(* Logix 5000 project; controller PBS_Perfusion vendor 1 type 14 code 217 rev 32.14; software revision 32.03; part 22 of 27 *)
(* tags used below, declared in another part *)
   Inp_SpeedFdbk : REAL;   // Speed Feedbak in Drive Units (typ. 0-32767 = 0 to max freq.)
   Inp_Datalink : REAL;   // Auxiliary Signal (datalink) Input in Drive (raw) Units
   Inp_Ready : BOOL;   // 1=Drive is ready to run
   Inp_Running : BOOL;   // 1=Drive is Running (active)
   Inp_CommandDir : BOOL;   // 1=Drive is commanded Forward, 0=Drive is commanded Reverse
   Inp_ActualDir : BOOL;   // 1=Drive is running Forward, 0=Drive is running Reverse
   Inp_Accelerating : BOOL;   // 1=Drive is accelerating
   Inp_Decelerating : BOOL;   // 1=Drive is decelerating
   Inp_Alarm : BOOL;   // 1=Drive has an Alarm Condition (see drive display or manual)
   Inp_Faulted : BOOL;   // 1=Drive has Faulted (see drive display or manual)
   Inp_AtSpeed : BOOL;   // 1=Drive is at commanded speed
   Inp_FwdPermOK : BOOL;   // 1=Permissives OK, drive can start Forward
   Inp_FwdNBPermOK : BOOL;   // 1=Non-Bypassable Permissives OK, drive can start Forward
   Inp_RevPermOK : BOOL;   // 1=Permissives OK, drive can start Reverse
   Inp_RevNBPermOK : BOOL;   // 1=Non-Bypassable Permissives OK, motor can start Reverse
   Inp_IntlkOK : BOOL;   // 1=Interlocks OK, drive can start/run
   Inp_NBIntlkOK : BOOL;   // 1=Non-Bypassable Interlocks OK, drive can start/run
   Inp_IntlkAvail : BOOL;   // 1 = Interlock Availibility OK
   Inp_IOFault : BOOL;   // Input Communication Status 0=OK, 1=fail
   Inp_Sim : BOOL;   // 1=Simulate working drive; 0=Start/Stop/ Monitor actual drive
   Inp_OvrdCmd : DINT;   // Override Command: 0=None, 1=Stop, 2=Start Fwd 3=Start Rev
   Inp_OvrdSpeed : REAL;   // Value to set Speed Reference in Override Mode (SpeedRef EU)
   Inp_OvrdOutDatalink : REAL;   // Value to set Output Datalink in Override Mode (OutDatalink EU)
   Inp_Reset : BOOL;   // 1=Reset Shed Latches and Cleared Alarms
   Cfg_HasReverse : BOOL;   // 1=Drive can be run reverse, 0=Forward only
   Cfg_HasJog : BOOL;   // 1=Drive Jog Command enabled/visible, 0=Drive Jog Command not allowed
   Cfg_AllowLocal : BOOL;   // 1=Allow Local Start/Stop without alarm, 0=Start/Stop from HMI/prog only
   Cfg_HasRunFdbk : BOOL;   // 1=Drive provides feedback signal on Inp_Running when running
   Cfg_UseRunFdbk : BOOL;   // 1=Drive run feedback should be used for failure checking
   Cfg_HasSpeedFdbk : BOOL;   // 1=Drive provides speed feedback on Inp_SpeedFdbk
   Cfg_UseSpeedFdbk : BOOL;   // 1=Drive speed determines running state, 0=state determined by drive Active input bit
   Cfg_HasInpDatalink : BOOL;   // 1=A signal is connected to Inp_Datalink
   Cfg_SetTrack : BOOL;   // 1=Settings track for unselected sources, 0=no tracking
   Cfg_SetTrackOvrdHand : BOOL;   // 1=Prog/Oper/Ext Settings track Override/Hand
   Cfg_OperStopPrio : BOOL;   // 1=OCmd_Stop any time, 0=OCmd_Stop only when Oper selected
   Cfg_ExtStopPrio : BOOL;   // 1=XCmd_Stop any time, 0=XCmd_Stop only when Ext selected
   Cfg_OCmdResets : BOOL;   // 1=New drive OCmd resets shed latches and cleared alarms, 0=OCmdReset req'd.
   Cfg_XCmdResets : BOOL;   // 1=New drive XCmd resets shed latches and cleared alarms, 0=XCmdReset req'd.
   Cfg_OvrdPermIntlk : BOOL;   // 1=Override ignores Bypassable Perm/ Intlk; 0=always use Perm/Intlk
   Cfg_ShedOnIOFault : BOOL;   // 1=Stop Motor and Alarm on I/O Fault; 0=Alarm only on I/O Fault
   Cfg_SimScaleEU : BOOL;   // 1=In simulation, scale Speed Ref EU to Speed Fdbk EU
   Cfg_SimScaleRaw : BOOL;   // 1=In simulation, scale Speed Ref EU to raw, then raw to Speed Fdbk EU
   Cfg_MaxSpdRef : REAL;   // Maximum Speed Reference in EU (for limiting)
   Cfg_SpeedRefRawMin : REAL;   // Speed Reference Minimum in Drive (raw) Units (for scaling)
   Cfg_SpeedRefRawMax : REAL;   // Speed Reference Maximum in Drive (raw) Units (for scaling)
   Cfg_SpeedRefEUMin : REAL;   // Speed Reference Minimum in Engineering Units (for scaling)
   Cfg_SpeedRefEUMax : REAL;   // Speed Reference Maximum in Engineering Units (for scaling)
   Cfg_SpeedFdbkRawMin : REAL;   // Speed Feedback Minimum in Drive (raw) Units (for scaling)
   Cfg_SpeedFdbkRawMax : REAL;   // Speed Feedback Maximum in Drive (raw) Units (for scaling)
   Cfg_SpeedFdbkEUMin : REAL;   // Speed Feedback Minimum in Engineering Units (for scaling)
   Cfg_SpeedFdbkEUMax : REAL;   // Speed Feedback Maximum in Engineering Units (for scaling)
   Cfg_InpDatalinkRawMin : REAL;   // Input Datalink Minimum in Drive (raw) Units (for scaling)
   Cfg_InpDatalinkRawMax : REAL;   // Input Datalink Maximum in Drive (raw) Units (for scaling)
   Cfg_InpDatalinkEUMin : REAL;   // Input Datalink Minimum in Engineering Units (for scaling)
   Cfg_InpDatalinkEUMax : REAL;   // Input Datalink Maximum in Engineering Units (for scaling)
   Cfg_OutDatalinkMin : REAL;   // Minimum Output Datalink in EU (for limiting)
   Cfg_OutDatalinkMax : REAL;   // Maximum Output Datalink in EU (for limiting)
   Cfg_SimRampT : REAL;   // Time to ramp speed fdbk when in Simulation (sec)
   PSet_SpeedRef : REAL;   // Program Setting of Speed Reference (EU)
   PSet_OutDatalink : REAL;   // Program Setting of Output Datalink (EU)
   XSet_SpeedRef : REAL;   // External Setting of Speed Reference (EU)
   XSet_OutDatalink : REAL;   // External Setting of Output Datalink (EU)
   PCmd_StartFwd : BOOL;   // Program Command to Start Drive Forward
   PCmd_StartRev : BOOL;   // Program Command to Start Drive Reverse
   PCmd_Stop : BOOL;   // Program Command to Stop Drive
   PCmd_Reset : BOOL;   // Program Command to Reset drive fault and all Alarms requiring Reset
   PCmd_FailToStartAck : ALIAS FOR FailToStart.PCmd_Ack;   // Program Command to Acknowledge Fail to Start Alarm
   PCmd_FailToStopAck : ALIAS FOR FailToStop.PCmd_Ack;   // Program Command to Acknowledge Fail to Stop Alarm
   PCmd_IntlkTripAck : ALIAS FOR IntlkTrip.PCmd_Ack;   // Program Command to Acknowledge Interlock Trip Alarm
   PCmd_DriveFaultAck : ALIAS FOR DriveFault.PCmd_Ack;   // Program Command to Acknowledge Drive Fault Alarm
   PCmd_IOFaultAck : ALIAS FOR IOFault.PCmd_Ack;   // Program Command to Acknowledge I/O Fault Alarm
   XCmd_StartFwd : BOOL;   // External Command to Start Drive Forward
   XCmd_StartRev : BOOL;   // External Command to Start Drive Reverse
   XCmd_Stop : BOOL;   // External Command to Stop Drive
   XCmd_JogFwd : BOOL;   // External Command to Jog Drive Forward
   XCmd_JogRev : BOOL;   // External Command to Jog Drive Reverse
   XCmd_Reset : BOOL;   // Ext Cmd to clear shed latches and cleared alarms
   Out_ClearFault : BOOL;   // 1=Attempt to clear Drive Fault
   Val_SpeedFdbk : REAL;   // Speed Feedback (actual) from drive
   Val_InpDatalink : REAL;   // Input Datalink value from drive
   Val_SpeedFdbkEUMin : REAL;   // Minimum of Speed Feedback = MIN (Cfg_SpeedFdbkEUMin, Cfg_SpeedFdbkEUMax)
   Val_SpeedFdbkEUMax : REAL;   // Maximum of Speed Feedback = MAX (Cfg_SpeedFdbkEUMin, Cfg_SpeedFdbkEUMax)
   Val_Fdbk : DINT;   // Device Feedback 0=Stopped, 1=Running Fwd 2=Running Rev 3=Accelerating 4=Decelerating
   Sts_StartingFwd : BOOL;   // 1=Drive requested to run forward and awaiting run feedback
   Sts_StartingRev : BOOL;   // 1=Drive requested to run reverse and awaiting run feedback
   Sts_RunningFwd : BOOL;   // 1=Drive requested to run and is confirmed running forward
   Sts_RunningRev : BOOL;   // 1=Drive requested to run and is confirmed running reverse
   Sts_CommandDir : BOOL;   // 1=Drive commanded to Forward, 0=Reverse
   Sts_ActualDir : BOOL;   // 1=Drive Actual direction is Forward, 0=Reverse
   Sts_Accel : BOOL;   // 1=Drive is Accelerating
   Sts_Decel : BOOL;   // 1=Drive is Decelerating
   Sts_NotReady : BOOL;   // 1=Drive is Not Ready (cannot be started) Check alarms, stops, faults
   Sts_Alarm : BOOL;   // 1=Drive has an Alarm (see drive display or manual)
   Sts_AtSpeed : BOOL;   // 1=Drive is running at reference speed
   Sts_Available : BOOL;   // 1=Drive available for control by automation (Prog)
   Sts_Bypass : BOOL;   // 1=Bypassable Interlocks and Permissives are Bypassed
   Sts_BypActive : BOOL;   // 1=Bypassing Active (Bypassed or Maintenance)
   Sts_NotRdy : BOOL;   // 1=Device Not Ready, see detail bits for reason
   Nrdy_CfgErr : BOOL;   // 1=Device Not Ready: Configuration Error
   Nrdy_DriveNR : BOOL;   // 1=Device Note Ready: Drive Not Ready
   Nrdy_Fail : BOOL;   // 1=Device Not Ready: Device Failure (Shed Requires Reset)
   Nrdy_Intlk : BOOL;   // 1=Device Not Ready: Interlock Not OK
   Nrdy_IOFault : BOOL;   // 1=Device Not Ready: I/O Fault (Shed Requires Reset)
   Nrdy_OoS : BOOL;   // 1=Device Not Ready: Device is Out of Service
   Nrdy_Perm : BOOL;   // 1=Device Not Ready: Permissive Not OK
   Nrdy_PrioStop : BOOL;   // 1=Device Not Ready: Oper/Ext Priority Stop Requires Reset
   Nrdy_Trip : BOOL;   // 1=Device not Ready: Deivce Tripped (Drive Fault)
   Sts_MaintByp : BOOL;   // 1=A Maintenance Bypass is Active, display icon
   Err_FdbkRaw : BOOL;   // 1=Erron in Config: Speed Fdbk Raw Min = Max
   Err_FdbkEU : BOOL;   // 1=Error in Config: Speed Fdbk EU Min = Max
   Err_RefEU : BOOL;   // 1=Error in Config: Speed Ref EU Min = Max
   Err_InpDLEU : BOOL;   // 1=Error in Config: Input Datalink EU Min = Max
   Sts_Hand : ALIAS FOR CmdSrc.Sts_Hand;
   Sts_OoS : ALIAS FOR CmdSrc.Sts_OoS;
   Sts_Maint : ALIAS FOR CmdSrc.Sts_Maint;
   Sts_Ovrd : ALIAS FOR CmdSrc.Sts_Ovrd;
   Sts_Prog : ALIAS FOR CmdSrc.Sts_Prog;
   Sts_Oper : ALIAS FOR CmdSrc.Sts_Oper;
   Sts_FailToStart : ALIAS FOR FailToStart.Inp;   // 1=Drive Failed to Start (One-Shot)
   Sts_FailToStop : ALIAS FOR FailToStop.Inp;   // 1=Drive Failed to Stop
   Sts_IntlkTrip : ALIAS FOR IntlkTrip.Inp;   // 1=Drive was stopped by an Interlock NOT OK (One-Shot)
   Sts_DriveFault : ALIAS FOR DriveFault.Inp;   // 1=Drive Fault (see drive display or manual)
   Sts_IOFault : ALIAS FOR IOFault.Inp;   // I/O Comm Fault Status (0=OK, 1=Bad)
   P_VSD : BOOL;   // Unique Parameter Name for auto - discovery
   CmdSrc : P_CmdSrc;   // Drive Mode Selection
   IOFault : P_Alarm;   // I/O Fault Alarm
   IntlkTrip : P_Alarm;   // Interlock Trip Alarm
   FailToStop : P_Alarm;   // Drive Failed to Stop Alarm
   FailToStart : P_Alarm;   // Drive Failed to Start Alarm
   Wrk_Run : BOOL;   // 1=Drive should be "running", 0=should be "stopped"
   Wrk_StartRetrigT : TIMER;   // Time to pulse start output on start command retrigger (Maint)
   Wrk_StopRetrigT : TIMER;   // Time to pulse stop output on stop command retrigger (Maint)
   Wrk_RunFdbk : BOOL;   // Run Feedback based on mode, simulation, etc. 1=running
   Wrk_Bypass : BOOL;   // Internal Bypassable Permissives and Interlocks are Bypassed flag
   DriveFault : P_Alarm;   // Drive Faulted Alarm
   Wrk_SpeedRef : REAL;   // Working copy of Speed Reference (for limiting)
   Wrk_Rev : BOOL;   // Working (internal) Direction 1=Reverse 0=Forward (default)
   Wrk_Jog : BOOL;   // 1=Jog Drive, 0=Drive not jogging
   Wrk_ResetT : TIMER;   // Reset Output Pulse Timer
   Wrk_ResetONS : BOOL;   // One-Shot to fire Reset Timer to ensure min. output ON time.
   Wrk_OutDatalink : REAL;   // Selected Output Datalink setting
   Wrk_StopT : TIMER;   // Stop Check Timer (for Fail to Stop)
   Wrk_StartT : TIMER;   // Start Check Timer (for Fail to Start)
   Wrk_Retrigger : BOOL;   // Maint Start issued while running or Stop while stopped
   Wrk_Step : REAL;   // Amount to change simulated Speed Fdbk this scan (ramp)
   Wrk_ScanTime : REAL;   // Seconds since previous scan
   Wrk_ScanT : TIMER;   // Scan Timer (milliseconds, always runs)
   Wrk_SimFdbkTgt : REAL;   // Speed Ref converted to Speed Fdbk units for simulation: target speed fdbk
   Wrk_JogT : TIMER;   // Jog Timer
   Wrk_SimScaleEUONS : BOOL;   // Cfg_SimScaleEU became true this scan
   Wrk_SimScaleRawONS : BOOL;   // Cfg_SimScaleRaw became true this scan
   Wrk_NotRdyONS : BOOL;   // Assert Stop on One-Shot of Sts_NotRdy
   Wrk_NotRdy : BOOL;   // Device Not Ready conditions excluding shed latches
   Wrk_StartInhT : TIMER;   // Local Start Inhibit Timer
   Wrk_StopInhT : TIMER;   // Local Stop Inhibit Timer
   Wrk_NoLongerSim : BOOL;   // Switched from Simulated to Real Drive this scan
   Wrk_Hand : BOOL;   // Perform Hand Mode alignment with actual device state
   Wrk_StartHornT : TIMER;   // Timer for audible alert or start
   Wrk_StartHorn : BOOL;   // 1=Sound audible prior to commanded motor start
   Wrk_RevPermOK : BOOL;   // Reverse Permissives and NB Permissive OK
   Wrk_FwdPermOK : BOOL;   // Forward Permissives and NB Permissive OK
   OCmd_ResetAckAll : BOOL;   // Oper Cmd to reset shed latches and cleared alarms, plus Acknowledge alarms
   OCmd_Reset : BOOL;   // Oper Cmd to clear shed latches and cleared alarms
   OCmd_JogRev : BOOL;   // Operator Command to Jog Drive Reverse (not cleared by instruction!)
   OCmd_JogFwd : BOOL;   // Operator Command to Jog Drive Forward (not cleared by instruction!)
   OCmd_Stop : BOOL;   // Operator Command to Stop Drive
   OCmd_StartRev : BOOL;   // Operator Command to Start Drive Reverse
   OCmd_StartFwd : BOOL;   // Operator Command to Start Drive Forward
   MCmd_Check : BOOL;   // Maintenance Command to Check (not bypass) all Interlocks and Permissives
   MCmd_Bypass : BOOL;   // Maintenance Command to Bypass all Bypassable Interlocks and Permissives
   OSet_OutDatalink : REAL;   // Operator Setting of Output Datalink (EU)
   OSet_SpeedRef : REAL;   // Operator Setting of Speed Reference (EU)
   ORdy_OSet : BOOL;   // 1=Ready for OSets (other than Speed Ref) (enables data entry fields)
   ORdy_SpeedRef : BOOL;   // 1=Ready for OSet_SpeedRef (enables data entry field)
   MRdy_Check : BOOL;   // 1=Ready for MCmd_Check (enables HMI button)
   MRdy_Bypass : BOOL;   // 1=Ready for MCmd_Bypass (enables HMI button)
   Wrk_ExtHas3 : BOOL;   // External has Output Datalink
   Wrk_ExtHas1 : BOOL;   // External has Commands
   Wrk_ExtHas0 : BOOL;   // External has Speed Reference
   Wrk_ProgHas3 : BOOL;   // Program has Output Datalink
   Wrk_ProgHas1 : BOOL;   // Program has Commands
   Wrk_ProgHas0 : BOOL;   // Program has Speed Reference
   Wrk_OperHas3 : BOOL;   // Operator has Output Datalink
   Wrk_OperHas1 : BOOL;   // Operator has Commands
   Wrk_OperHas0 : BOOL;   // Operator has Speed Reference
   ONS : DINT[3];
   REAL : DINT;
(* P_VSD, continued *)

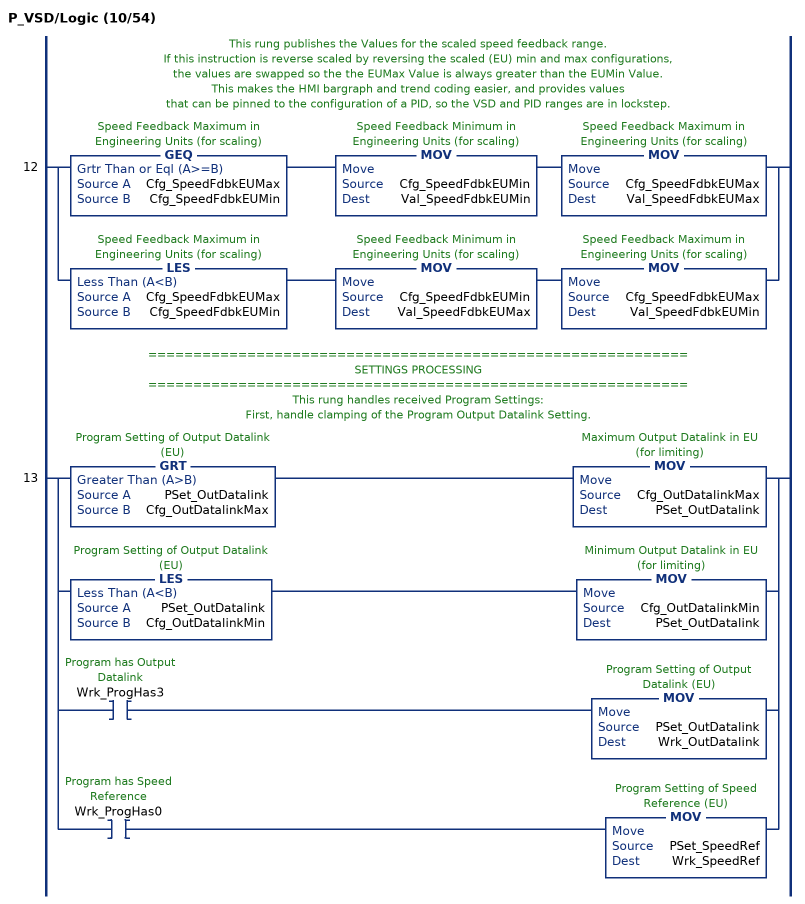
   [picture p487: P_VSD/Logic rungs 12-13]
   // This rung publishes the Values for the scaled speed feedback range.
   // If this instruction is reverse scaled by reversing the scaled (EU) min and max configurations,
   // the values are swapped so the the EUMax Value is always greater than the EUMin Value.
   // This makes the HMI bargraph and trend coding easier, and provides values
   // that can be pinned to the configuration of a PID, so the VSD and PID ranges are in lockstep.
   12: [GEQ(Cfg_SpeedFdbkEUMax,Cfg_SpeedFdbkEUMin) MOV(Cfg_SpeedFdbkEUMin,Val_SpeedFdbkEUMin) MOV(Cfg_SpeedFdbkEUMax,Val_SpeedFdbkEUMax) ,LES(Cfg_SpeedFdbkEUMax,Cfg_SpeedFdbkEUMin) MOV(Cfg_SpeedFdbkEUMin,Val_SpeedFdbkEUMax) MOV(Cfg_SpeedFdbkEUMax,Val_SpeedFdbkEUMin) ];
   // ============================================================
   // SETTINGS PROCESSING
   // ============================================================
   // This rung handles received Program Settings:
   // First, handle clamping of the Program Output Datalink Setting.
   13: [GRT(PSet_OutDatalink,Cfg_OutDatalinkMax) MOV(Cfg_OutDatalinkMax,PSet_OutDatalink) ,LES(PSet_OutDatalink,Cfg_OutDatalinkMin) MOV(Cfg_OutDatalinkMin,PSet_OutDatalink) ,XIC(Wrk_ProgHas3) MOV(PSet_OutDatalink,Wrk_OutDatalink) ,XIC(Wrk_ProgHas0) MOV(PSet_SpeedRef,Wrk_SpeedRef) ];
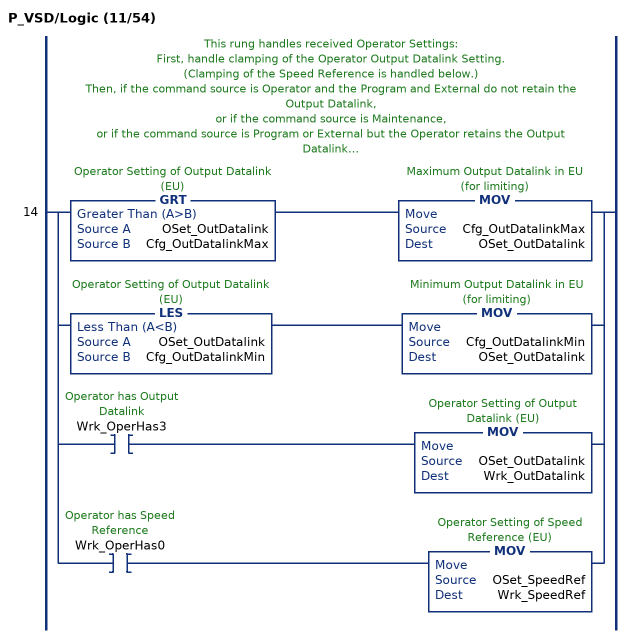
   // This rung handles received Operator Settings:
   // First, handle clamping of the Operator Output Datalink Setting.
   // (Clamping of the Speed Reference is handled below.)
   // Then, if the command source is Operator and the Program and External do not retain the Output Datalink,
   // or if the command source is Maintenance,
   // or if the command source is Program or External but the Operator retains the Output Datalink,
   // use the Operator Setting for the Output Datalink.
   // The Operator Setting for the Speed Reference is handled similarly.
   // #####  Changed P_Mode to P_CmdSrc. Added External Command Source and Commands.  #####
   14: [GRT(OSet_OutDatalink,Cfg_OutDatalinkMax) MOV(Cfg_OutDatalinkMax,OSet_OutDatalink) ,LES(OSet_OutDatalink,Cfg_OutDatalinkMin) MOV(Cfg_OutDatalinkMin,OSet_OutDatalink) ,XIC(Wrk_OperHas3) MOV(OSet_OutDatalink,Wrk_OutDatalink) ,XIC(Wrk_OperHas0) MOV(OSet_SpeedRef,Wrk_SpeedRef) ];
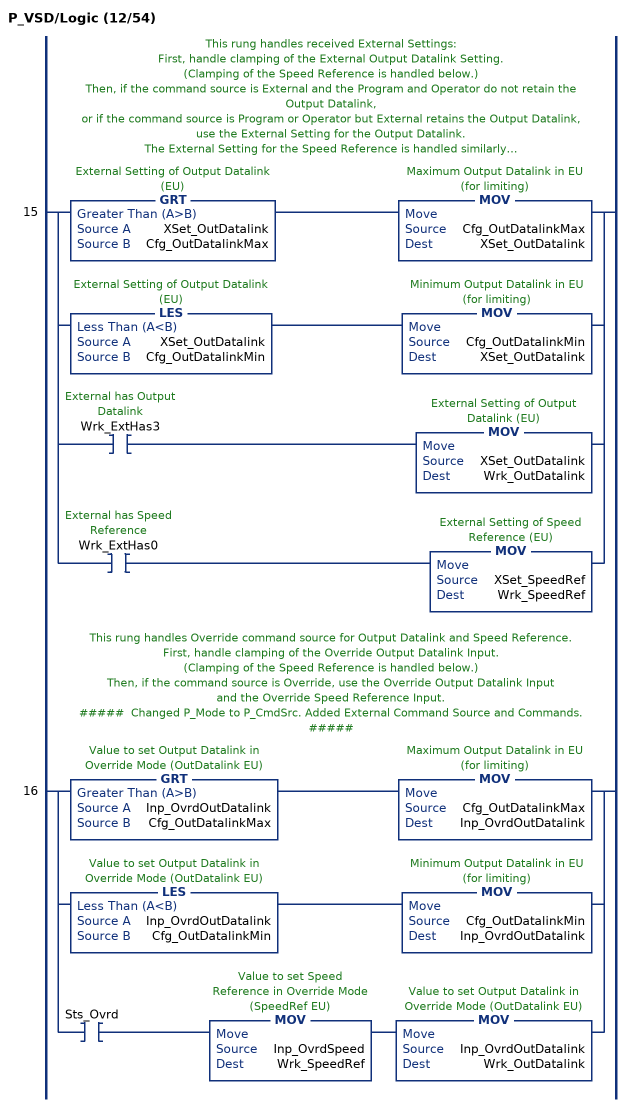
   // This rung handles received External Settings:
   // First, handle clamping of the External Output Datalink Setting.
   // (Clamping of the Speed Reference is handled below.)
   // Then, if the command source is External and the Program and Operator do not retain the Output Datalink,
   // or if the command source is Program or Operator but External retains the Output Datalink,
   // use the External Setting for the Output Datalink.
   // The External Setting for the Speed Reference is handled similarly.
   // #####  Changed P_Mode to P_CmdSrc. Added External Command Source and Commands.  #####
   15: [GRT(XSet_OutDatalink,Cfg_OutDatalinkMax) MOV(Cfg_OutDatalinkMax,XSet_OutDatalink) ,LES(XSet_OutDatalink,Cfg_OutDatalinkMin) MOV(Cfg_OutDatalinkMin,XSet_OutDatalink) ,XIC(Wrk_ExtHas3) MOV(XSet_OutDatalink,Wrk_OutDatalink) ,XIC(Wrk_ExtHas0) MOV(XSet_SpeedRef,Wrk_SpeedRef) ];
   // This rung handles Override command source for Output Datalink and Speed Reference.
   // First, handle clamping of the Override Output Datalink Input.
   // (Clamping of the Speed Reference is handled below.)
   // Then, if the command source is Override, use the Override Output Datalink Input
   // and the Override Speed Reference Input.
   // #####  Changed P_Mode to P_CmdSrc. Added External Command Source and Commands.  #####
   16: [GRT(Inp_OvrdOutDatalink,Cfg_OutDatalinkMax) MOV(Cfg_OutDatalinkMax,Inp_OvrdOutDatalink) ,LES(Inp_OvrdOutDatalink,Cfg_OutDatalinkMin) MOV(Cfg_OutDatalinkMin,Inp_OvrdOutDatalink) ,XIC(Sts_Ovrd) MOV(Inp_OvrdSpeed,Wrk_SpeedRef) MOV(Inp_OvrdOutDatalink,Wrk_OutDatalink) ];
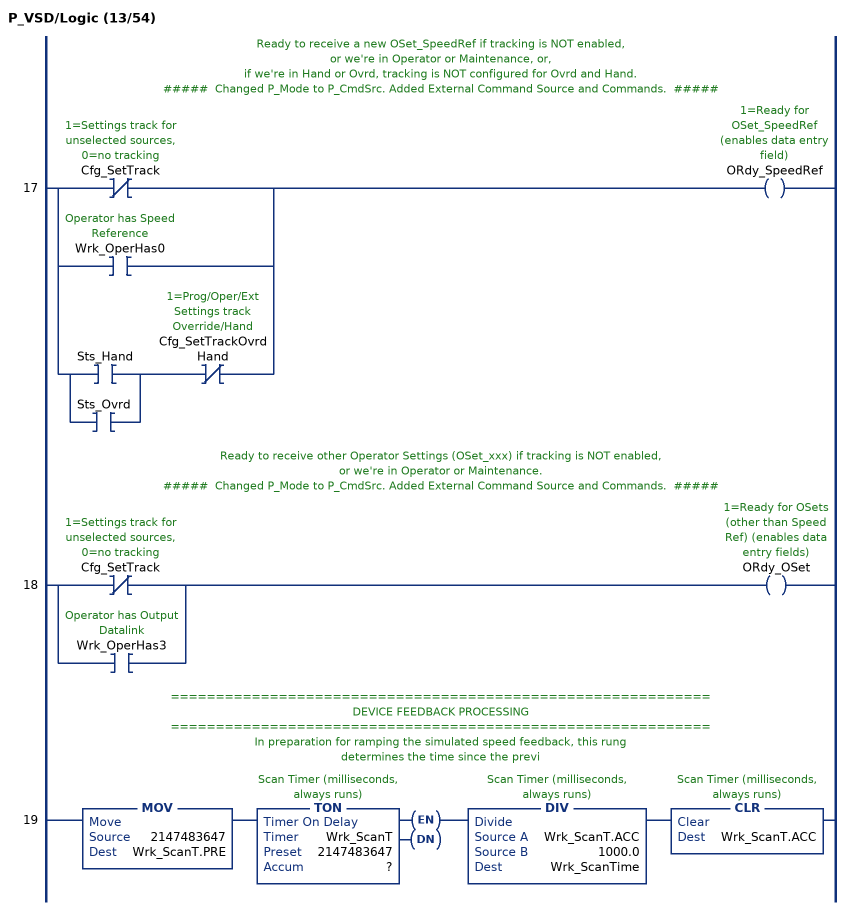
   // Ready to receive a new OSet_SpeedRef if tracking is NOT enabled,
   // or we're in Operator or Maintenance, or,
   // if we're in Hand or Ovrd, tracking is NOT configured for Ovrd and Hand.
   // #####  Changed P_Mode to P_CmdSrc. Added External Command Source and Commands.  #####
   17: [XIO(Cfg_SetTrack) ,XIC(Wrk_OperHas0) ,[XIC(Sts_Hand) ,XIC(Sts_Ovrd) ] XIO(Cfg_SetTrackOvrdHand) ]OTE(ORdy_SpeedRef);
   // Ready to receive other Operator Settings (OSet_xxx) if tracking is NOT enabled,
   // or we're in Operator or Maintenance.
   // #####  Changed P_Mode to P_CmdSrc. Added External Command Source and Commands.  #####
   18: [XIO(Cfg_SetTrack) ,XIC(Wrk_OperHas3) ]OTE(ORdy_OSet);
   // ============================================================
   // DEVICE FEEDBACK PROCESSING
   // ============================================================
   // In preparation for ramping the simulated speed feedback, this rung
   // determines the time since the previ
   19: MOV(2147483647,Wrk_ScanT.PRE)TON(Wrk_ScanT,?,?)DIV(Wrk_ScanT.ACC,1000.0,Wrk_ScanTime)CLR(Wrk_ScanT.ACC);
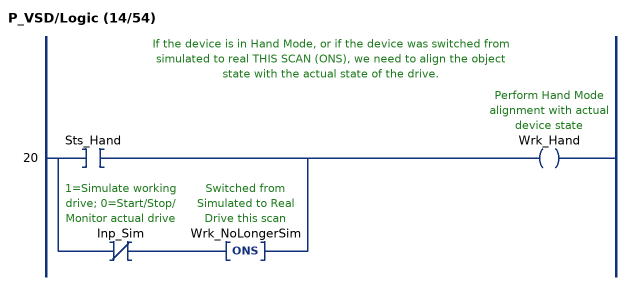
   // If the device is in Hand Mode, or if the device was switched from
   // simulated to real THIS SCAN (ONS), we need to align the object
   // state with the actual state of the drive.
   20: [XIC(Sts_Hand) ,XIO(Inp_Sim) ONS(Wrk_NoLongerSim) ]OTE(Wrk_Hand);
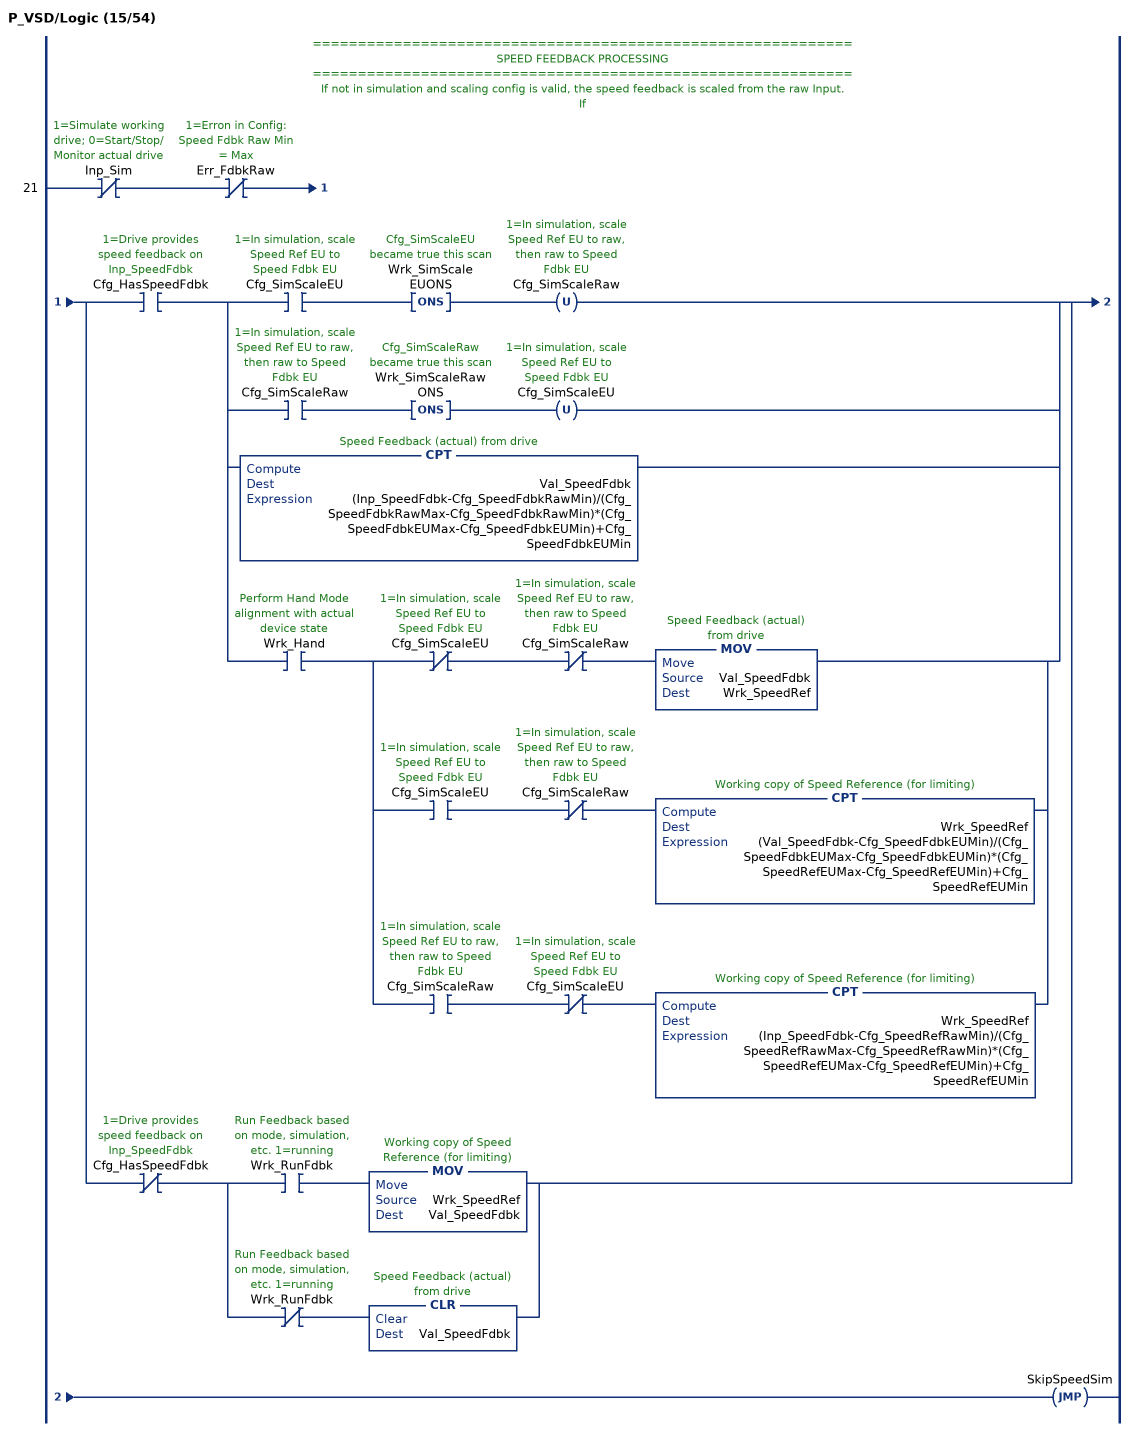
   // ============================================================
   // SPEED FEEDBACK PROCESSING
   // ============================================================
   // If not in simulation and scaling config is valid, the speed feedback is scaled from the raw Input.
   // If
   21: XIO(Inp_Sim)XIO(Err_FdbkRaw)[XIC(Cfg_HasSpeedFdbk) [XIC(Cfg_SimScaleEU) ONS(Wrk_SimScaleEUONS) OTU(Cfg_SimScaleRaw) ,XIC(Cfg_SimScaleRaw) ONS(Wrk_SimScaleRawONS) OTU(Cfg_SimScaleEU) ,CPT(Val_SpeedFdbk,(Inp_SpeedFdbk-Cfg_SpeedFdbkRawMin)/(Cfg_SpeedFdbkRawMax-Cfg_SpeedFdbkRawMin)*(Cfg_SpeedFdbkEUMax-Cfg_SpeedFdbkEUMin)+Cfg_SpeedFdbkEUMin) ,XIC(Wrk_Hand) [XIO(Cfg_SimScaleEU) XIO(Cfg_SimScaleRaw) MOV(Val_SpeedFdbk,Wrk_SpeedRef) ,XIC(Cfg_SimScaleEU) XIO(Cfg_SimScaleRaw) CPT(Wrk_SpeedRef,(Val_SpeedFdbk-Cfg_SpeedFdbkEUMin)/(Cfg_SpeedFdbkEUMax-Cfg_SpeedFdbkEUMin)*(Cfg_SpeedRefEUMax-Cfg_SpeedRefEUMin)+Cfg_SpeedRefEUMin) ,XIC(Cfg_SimScaleRaw) XIO(Cfg_SimScaleEU) CPT(Wrk_SpeedRef,(Inp_SpeedFdbk-Cfg_SpeedRefRawMin)/(Cfg_SpeedRefRawMax-Cfg_SpeedRefRawMin)*(Cfg_SpeedRefEUMax-Cfg_SpeedRefEUMin)+Cfg_SpeedRefEUMin) ] ] ,XIO(Cfg_HasSpeedFdbk) [XIC(Wrk_RunFdbk) MOV(Wrk_SpeedRef,Val_SpeedFdbk) ,XIO(Wrk_RunFdbk) CLR(Val_SpeedFdbk) ] ]JMP(SkipSpeedSim);
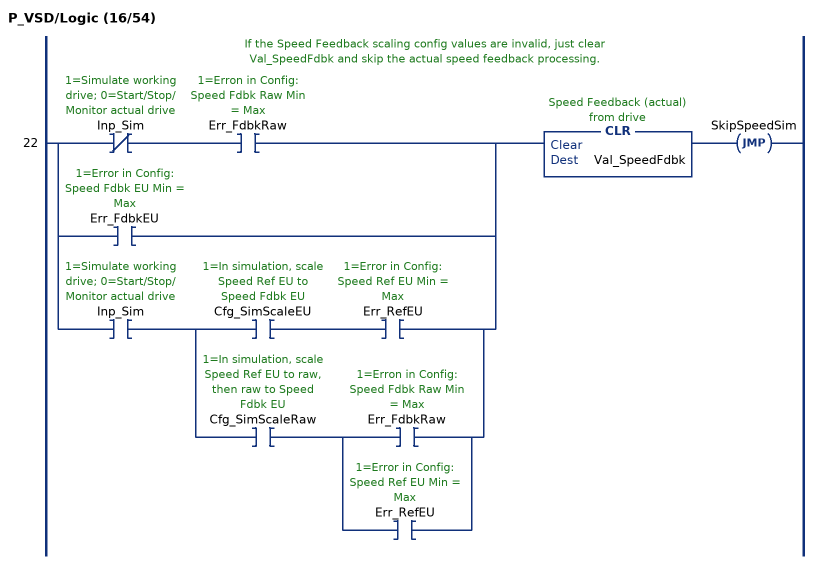
   // If the Speed Feedback scaling config values are invalid, just clear
   // Val_SpeedFdbk and skip the actual speed feedback processing.
   22: [XIO(Inp_Sim) XIC(Err_FdbkRaw) ,XIC(Err_FdbkEU) ,XIC(Inp_Sim) [XIC(Cfg_SimScaleEU) XIC(Err_RefEU) ,XIC(Cfg_SimScaleRaw) [XIC(Err_FdbkRaw) ,XIC(Err_RefEU) ] ] ]CLR(Val_SpeedFdbk)JMP(SkipSpeedSim);
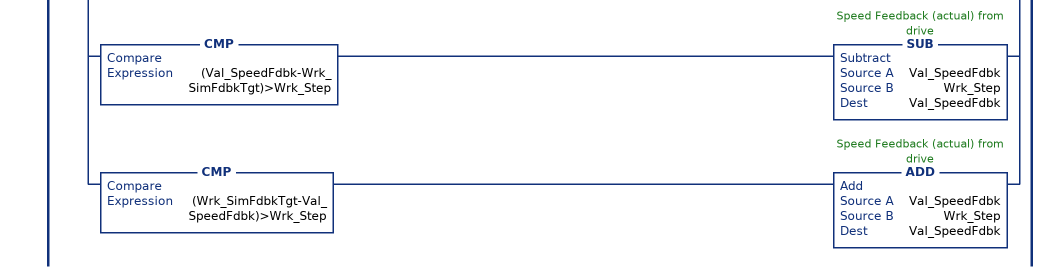
   // If in simulation, simulate accel/decel.
   // #####  V4.00.00  2018-07-13:  Changed delay / time configuration items to REAL seconds.  #####
   23: XIC(Inp_Sim)[[XIC(Wrk_Run) ,XIC(Wrk_Jog) ] [XIO(Cfg_SimScaleEU) XIO(Cfg_SimScaleRaw) MOV(Wrk_SpeedRef,Wrk_SimFdbkTgt) ,[XIC(Cfg_SimScaleEU) XIO(Cfg_SimScaleRaw) CPT(Wrk_SimFdbkTgt,(Wrk_SpeedRef-Cfg_SpeedRefEUMin)/(Cfg_SpeedRefEUMax-Cfg_SpeedRefEUMin)*(Cfg_SpeedFdbkEUMax-Cfg_SpeedFdbkEUMin)+Cfg_SpeedFdbkEUMin) ,XIC(Cfg_SimScaleRaw) [CPT(Wrk_SimFdbkTgt,(Wrk_SpeedRef-Cfg_SpeedRefEUMin)/(Cfg_SpeedRefEUMax-Cfg_SpeedRefEUMin)*(Cfg_SpeedRefRawMax-Cfg_SpeedRefRawMin)+Cfg_SpeedRefRawMin) ,CPT(Wrk_SimFdbkTgt,(Wrk_SimFdbkTgt-Cfg_SpeedFdbkRawMin)/(Cfg_SpeedFdbkRawMax-Cfg_SpeedFdbkRawMin)*(Cfg_SpeedFdbkEUMax-Cfg_SpeedFdbkEUMin)+Cfg_SpeedFdbkEUMin) ] ] ] ,[XIO(Wrk_Run) XIO(Wrk_Jog) ,XIO(Wrk_Rev) XIO(Sts_ActualDir) ,XIC(Wrk_Rev) XIC(Sts_ActualDir) ] CLR(Wrk_SimFdbkTgt) ,GRT(Cfg_SimRampT,0.0) [CPT(Wrk_Step,Cfg_MaxSpdRef/Cfg_SimRampT*Wrk_ScanTime) ,XIC(Cfg_SimScaleEU) XIO(Cfg_SimScaleRaw) CPT(Wrk_Step,(Wrk_Step-Cfg_SpeedRefEUMin)/(Cfg_SpeedRefEUMax-Cfg_SpeedRefEUMin)*(Cfg_SpeedFdbkEUMax-Cfg_SpeedFdbkEUMin)+Cfg_SpeedFdbkEUMin) ,XIC(Cfg_SimScaleRaw) [CPT(Wrk_Step,(Wrk_Step-Cfg_SpeedRefEUMin)/(Cfg_SpeedRefEUMax-Cfg_SpeedRefEUMin)*(Cfg_SpeedRefRawMax-Cfg_SpeedRefRawMin)+Cfg_SpeedRefRawMin) ,CPT(Wrk_Step,(Wrk_Step-Cfg_SpeedFdbkRawMin)/(Cfg_SpeedFdbkRawMax-Cfg_SpeedFdbkRawMin)*(Cfg_SpeedFdbkEUMax-Cfg_SpeedFdbkEUMin)+Cfg_SpeedFdbkEUMin) ] ] ,LEQ(Cfg_SimRampT,0.0) MOV(1.50000000e+038,Wrk_Step) ,CMP(ABS(Val_SpeedFdbk-Wrk_SimFdbkTgt)<=Wrk_Step) MOV(Wrk_SimFdbkTgt,Val_SpeedFdbk) ,CMP((Val_SpeedFdbk-Wrk_SimFdbkTgt)>Wrk_Step) SUB(Val_SpeedFdbk,Wrk_Step,Val_SpeedFdbk) ,CMP((Wrk_SimFdbkTgt-Val_SpeedFdbk)>Wrk_Step) ADD(Val_SpeedFdbk,Wrk_Step,Val_SpeedFdbk) ];
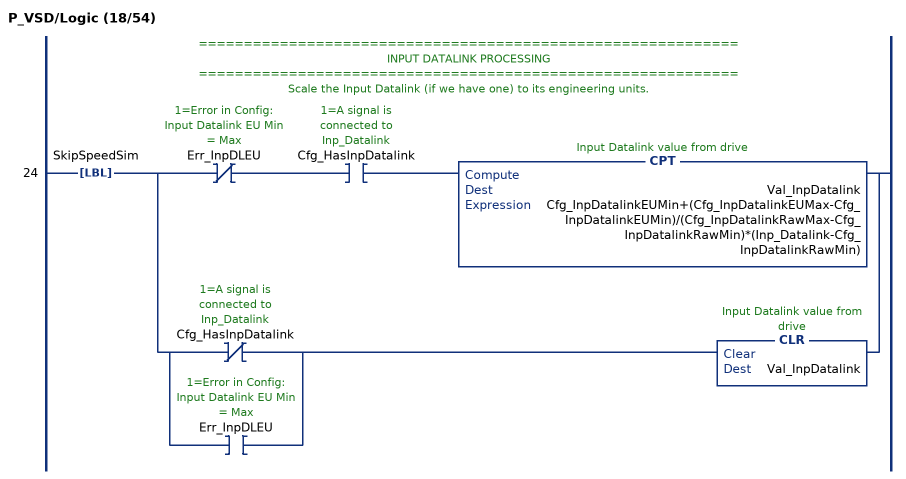
   // ============================================================
   // INPUT DATALINK PROCESSING
   // ============================================================
   // Scale the Input Datalink (if we have one) to its engineering units.
   24: LBL(SkipSpeedSim)[XIO(Err_InpDLEU) XIC(Cfg_HasInpDatalink) CPT(Val_InpDatalink,Cfg_InpDatalinkEUMin+(Cfg_InpDatalinkEUMax-Cfg_InpDatalinkEUMin)/(Cfg_InpDatalinkRawMax-Cfg_InpDatalinkRawMin)*(Inp_Datalink-Cfg_InpDatalinkRawMin)) ,[XIO(Cfg_HasInpDatalink) ,XIC(Err_InpDLEU) ] CLR(Val_InpDatalink) ];
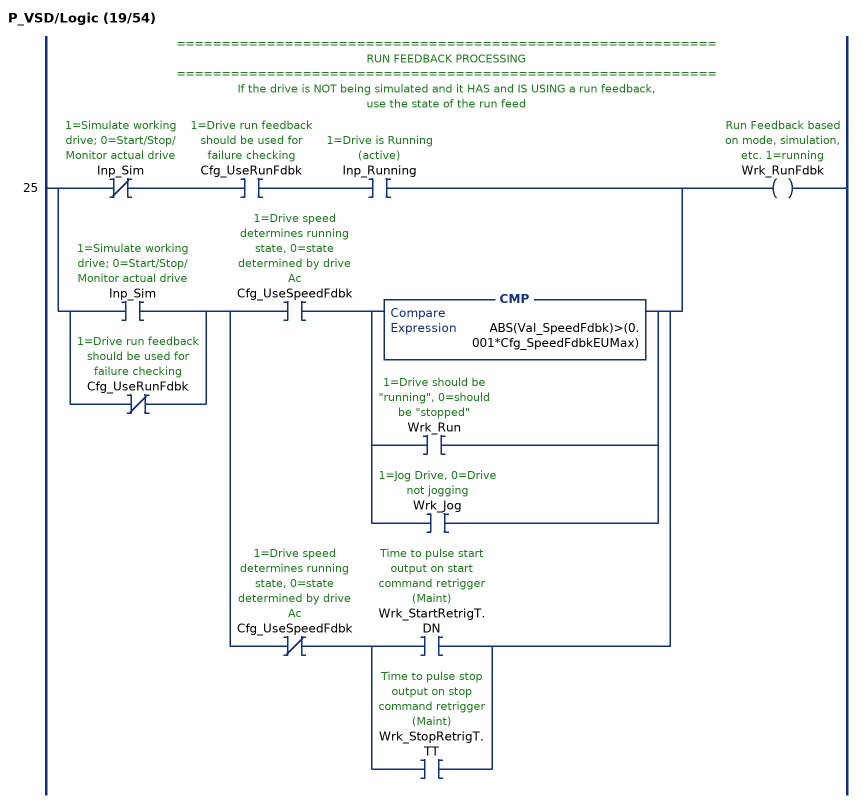
   // ============================================================
   // RUN FEEDBACK PROCESSING
   // ============================================================
   // If the drive is NOT being simulated and it HAS and IS USING a run feedback,
   // use the state of the run feed
   25: [XIO(Inp_Sim) XIC(Cfg_UseRunFdbk) XIC(Inp_Running) ,[XIC(Inp_Sim) ,XIO(Cfg_UseRunFdbk) ] [XIC(Cfg_UseSpeedFdbk) [CMP(ABS(Val_SpeedFdbk)>(0.001*Cfg_SpeedFdbkEUMax)) ,XIC(Wrk_Run) ,XIC(Wrk_Jog) ] ,XIO(Cfg_UseSpeedFdbk) [XIC(Wrk_StartRetrigT.DN) ,XIC(Wrk_StopRetrigT.TT) ] ] ]OTE(Wrk_RunFdbk);
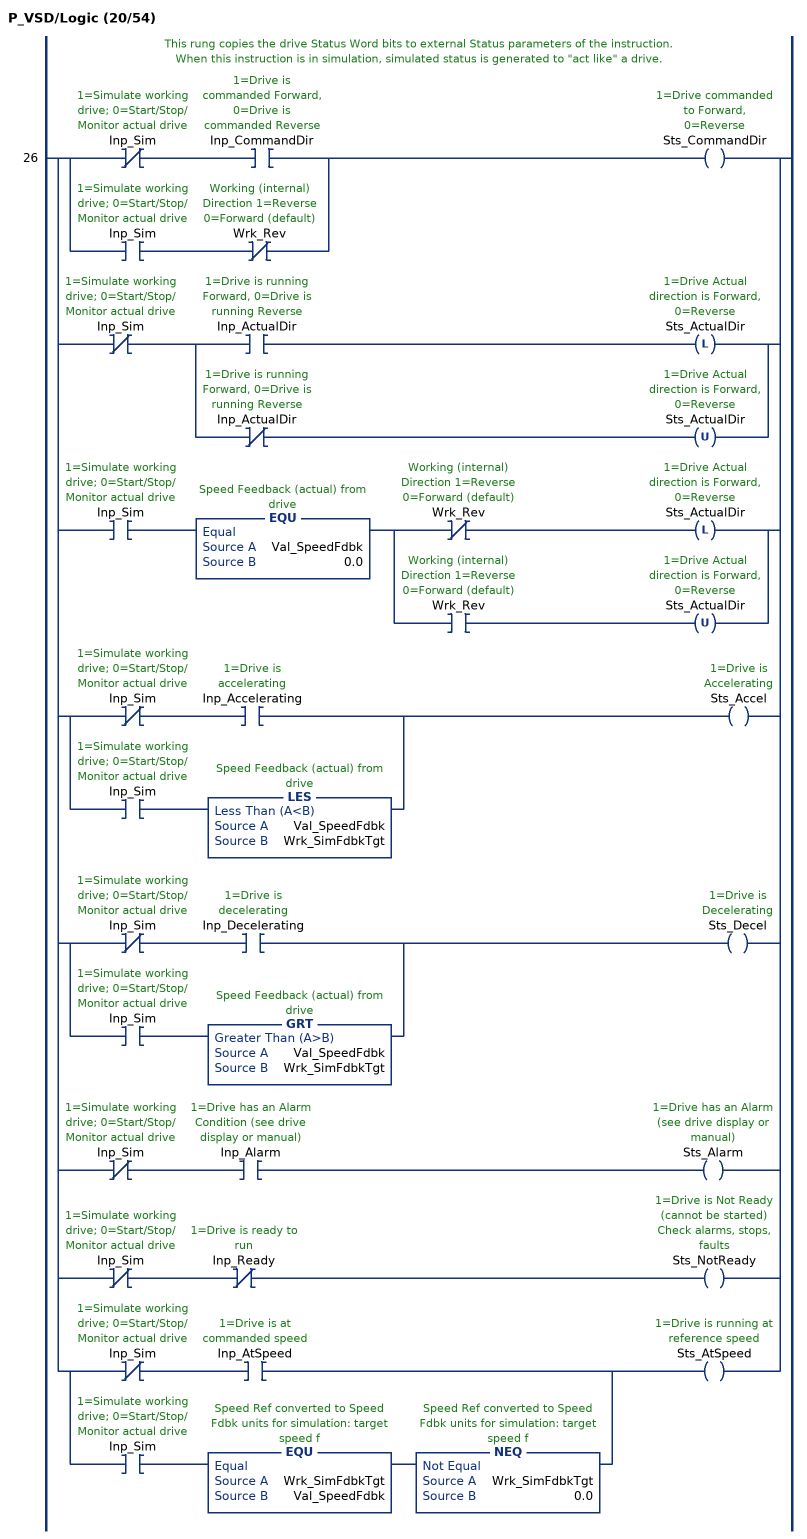
   // This rung copies the drive Status Word bits to external Status parameters of the instruction.
   // When this instruction is in simulation, simulated status is generated to "act like" a drive.
   26: [[XIO(Inp_Sim) XIC(Inp_CommandDir) ,XIC(Inp_Sim) XIO(Wrk_Rev) ] OTE(Sts_CommandDir) ,[XIO(Inp_Sim) [XIC(Inp_ActualDir) OTL(Sts_ActualDir) ,XIO(Inp_ActualDir) OTU(Sts_ActualDir) ] ,XIC(Inp_Sim) EQU(Val_SpeedFdbk,0.0) [XIO(Wrk_Rev) OTL(Sts_ActualDir) ,XIC(Wrk_Rev) OTU(Sts_ActualDir) ] ] ,[XIO(Inp_Sim) XIC(Inp_Accelerating) ,XIC(Inp_Sim) LES(Val_SpeedFdbk,Wrk_SimFdbkTgt) ] OTE(Sts_Accel) ,[XIO(Inp_Sim) XIC(Inp_Decelerating) ,XIC(Inp_Sim) GRT(Val_SpeedFdbk,Wrk_SimFdbkTgt) ] OTE(Sts_Decel) ,XIO(Inp_Sim) XIC(Inp_Alarm) OTE(Sts_Alarm) ,XIO(Inp_Sim) XIO(Inp_Ready) OTE(Sts_NotReady) ,[XIO(Inp_Sim) XIC(Inp_AtSpeed) ,XIC(Inp_Sim) EQU(Wrk_SimFdbkTgt,Val_SpeedFdbk) NEQ(Wrk_SimFdbkTgt,0.0) ] OTE(Sts_AtSpeed) ];
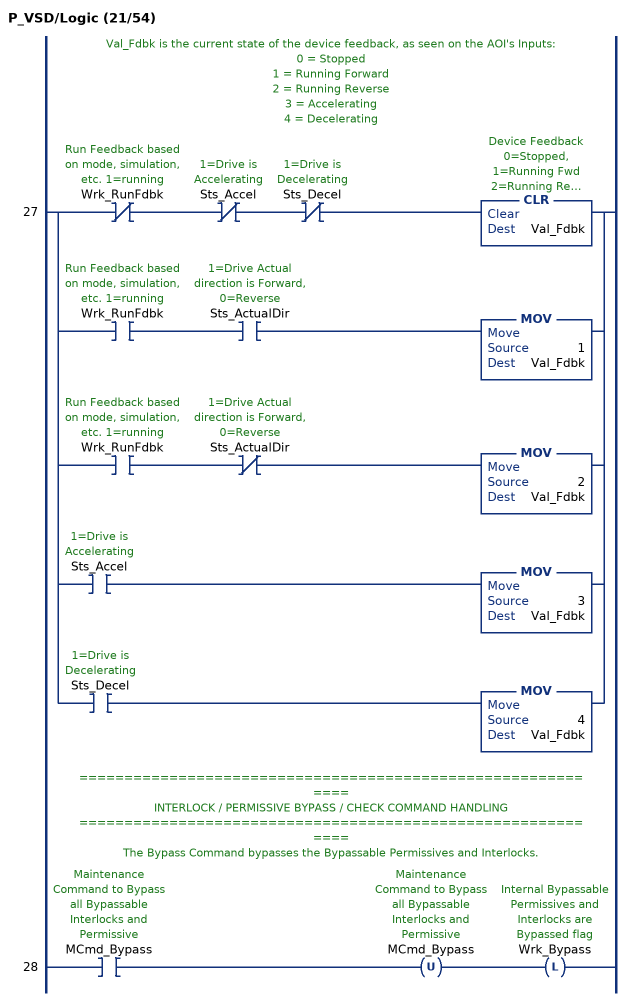
   // Val_Fdbk is the current state of the device feedback, as seen on the AOI's Inputs:
   // 0 = Stopped
   // 1 = Running Forward
   // 2 = Running Reverse
   // 3 = Accelerating
   // 4 = Decelerating
   27: [XIO(Wrk_RunFdbk) XIO(Sts_Accel) XIO(Sts_Decel) CLR(Val_Fdbk) ,XIC(Wrk_RunFdbk) XIC(Sts_ActualDir) MOV(1,Val_Fdbk) ,XIC(Wrk_RunFdbk) XIO(Sts_ActualDir) MOV(2,Val_Fdbk) ,XIC(Sts_Accel) MOV(3,Val_Fdbk) ,XIC(Sts_Decel) MOV(4,Val_Fdbk) ];
   // ============================================================
   // INTERLOCK / PERMISSIVE BYPASS / CHECK COMMAND HANDLING
   // ============================================================
   // The Bypass Command bypasses the Bypassable Permissives and Interlocks.
   28: XIC(MCmd_Bypass)OTU(MCmd_Bypass)OTL(Wrk_Bypass);
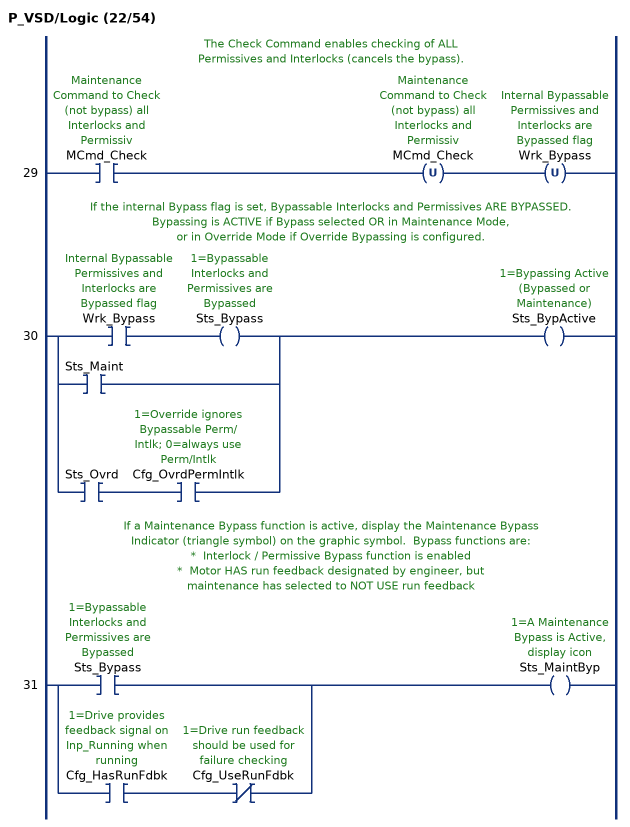
   // The Check Command enables checking of ALL
   // Permissives and Interlocks (cancels the bypass).
   29: XIC(MCmd_Check)OTU(MCmd_Check)OTU(Wrk_Bypass);
   // If the internal Bypass flag is set, Bypassable Interlocks and Permissives ARE BYPASSED.
   // Bypassing is ACTIVE if Bypass selected OR in Maintenance Mode,
   // or in Override Mode if Override Bypassing is configured.
   30: [XIC(Wrk_Bypass) OTE(Sts_Bypass) ,XIC(Sts_Maint) ,XIC(Sts_Ovrd) XIC(Cfg_OvrdPermIntlk) ]OTE(Sts_BypActive);
   // If a Maintenance Bypass function is active, display the Maintenance Bypass
   // Indicator (triangle symbol) on the graphic symbol.  Bypass functions are:
   // *  Interlock / Permissive Bypass function is enabled
   // *  Motor HAS run feedback designated by engineer, but
   // maintenance has selected to NOT USE run feedback
   31: [XIC(Sts_Bypass) ,XIC(Cfg_HasRunFdbk) XIO(Cfg_UseRunFdbk) ]OTE(Sts_MaintByp);
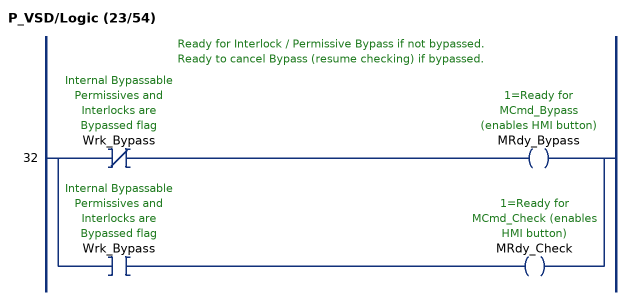
   // Ready for Interlock / Permissive Bypass if not bypassed.
   // Ready to cancel Bypass (resume checking) if bypassed.
   32: [XIO(Wrk_Bypass) OTE(MRdy_Bypass) ,XIC(Wrk_Bypass) OTE(MRdy_Check) ];
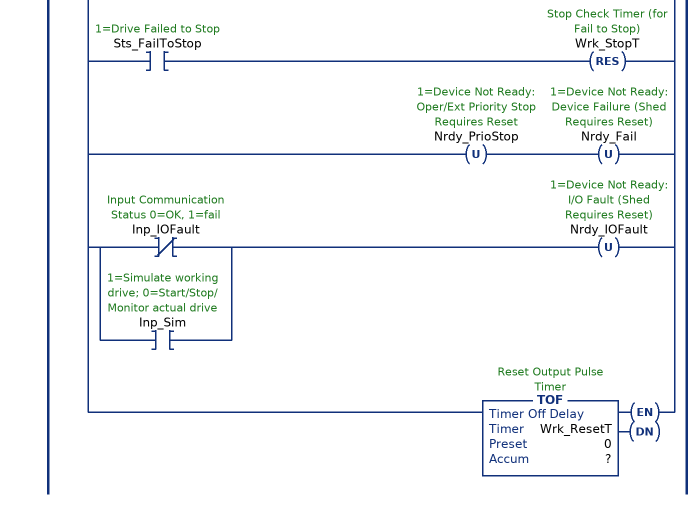
   // ============================================================
   // ALARM RESET COMMAND HANDLING
   // ============================================================
   // This rung handles the Alarm Reset Input and Commands
   // and the "Reset and Ack All" Operator Command.
   33: [XIC(OCmd_Reset) OTU(OCmd_Reset) ,XIC(XCmd_Reset) OTU(XCmd_Reset) ,XIC(PCmd_Reset) OTU(PCmd_Reset) ,XIC(Inp_Reset) ONS(Wrk_ResetONS) ,[XIC(OCmd_StartFwd) ,XIC(OCmd_StartRev) ,XIC(OCmd_Stop) ,[XIC(OCmd_JogFwd) ,XIC(OCmd_JogRev) ] XIC(Cfg_HasJog) ] XIC(Cfg_OCmdResets) XIC(Wrk_OperHas1) ,[XIC(XCmd_StartFwd) ,XIC(XCmd_StartRev) ,XIC(XCmd_Stop) ,[XIC(XCmd_JogFwd) ,XIC(XCmd_JogRev) ] XIC(Cfg_HasJog) ] XIC(Cfg_XCmdResets) XIC(Wrk_ExtHas1) ,XIC(OCmd_ResetAckAll) OTU(OCmd_ResetAckAll) [OTL(PCmd_FailToStartAck) ,OTL(PCmd_FailToStopAck) ,OTL(PCmd_DriveFaultAck) ,OTL(PCmd_IntlkTripAck) ,OTL(PCmd_IOFaultAck) ] ][OTL(FailToStart.PCmd_Reset) OTL(FailToStop.PCmd_Reset) OTL(IntlkTrip.PCmd_Reset) OTL(IOFault.PCmd_Reset) ,XIC(Sts_FailToStart) RES(Wrk_StartT) ,XIC(Sts_FailToStop) RES(Wrk_StopT) ,OTU(Nrdy_PrioStop) OTU(Nrdy_Fail) ,[XIO(Inp_IOFault) ,XIC(Inp_Sim) ] OTU(Nrdy_IOFault) ,TOF(Wrk_ResetT,?,?) ];
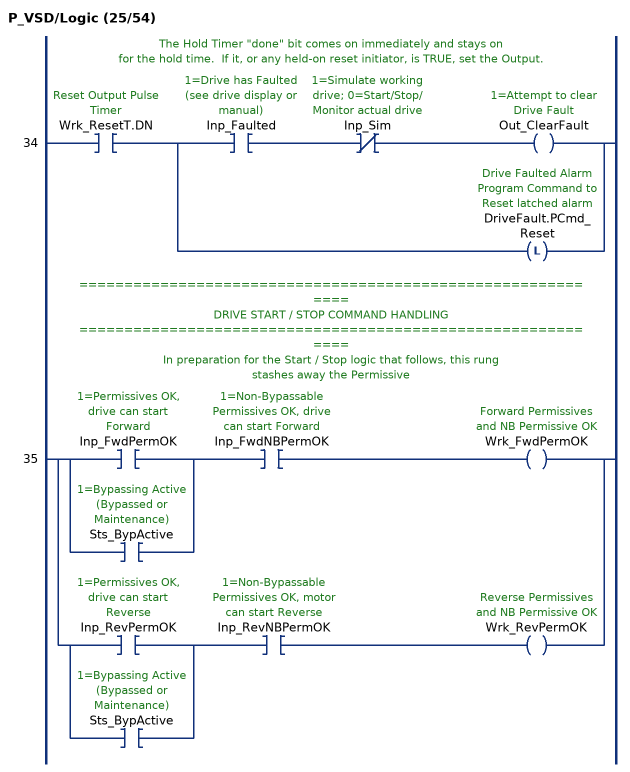
   // The Hold Timer "done" bit comes on immediately and stays on
   // for the hold time.  If it, or any held-on reset initiator, is TRUE, set the Output.
   34: XIC(Wrk_ResetT.DN)[XIC(Inp_Faulted) XIO(Inp_Sim) OTE(Out_ClearFault) ,OTL(DriveFault.PCmd_Reset) ];
   // ============================================================
   // DRIVE START / STOP COMMAND HANDLING
   // ============================================================
   // In preparation for the Start / Stop logic that follows, this rung
   // stashes away the Permissive
   35: [[XIC(Inp_FwdPermOK) ,XIC(Sts_BypActive) ] XIC(Inp_FwdNBPermOK) OTE(Wrk_FwdPermOK) ,[XIC(Inp_RevPermOK) ,XIC(Sts_BypActive) ] XIC(Inp_RevNBPermOK) OTE(Wrk_RevPermOK) ];
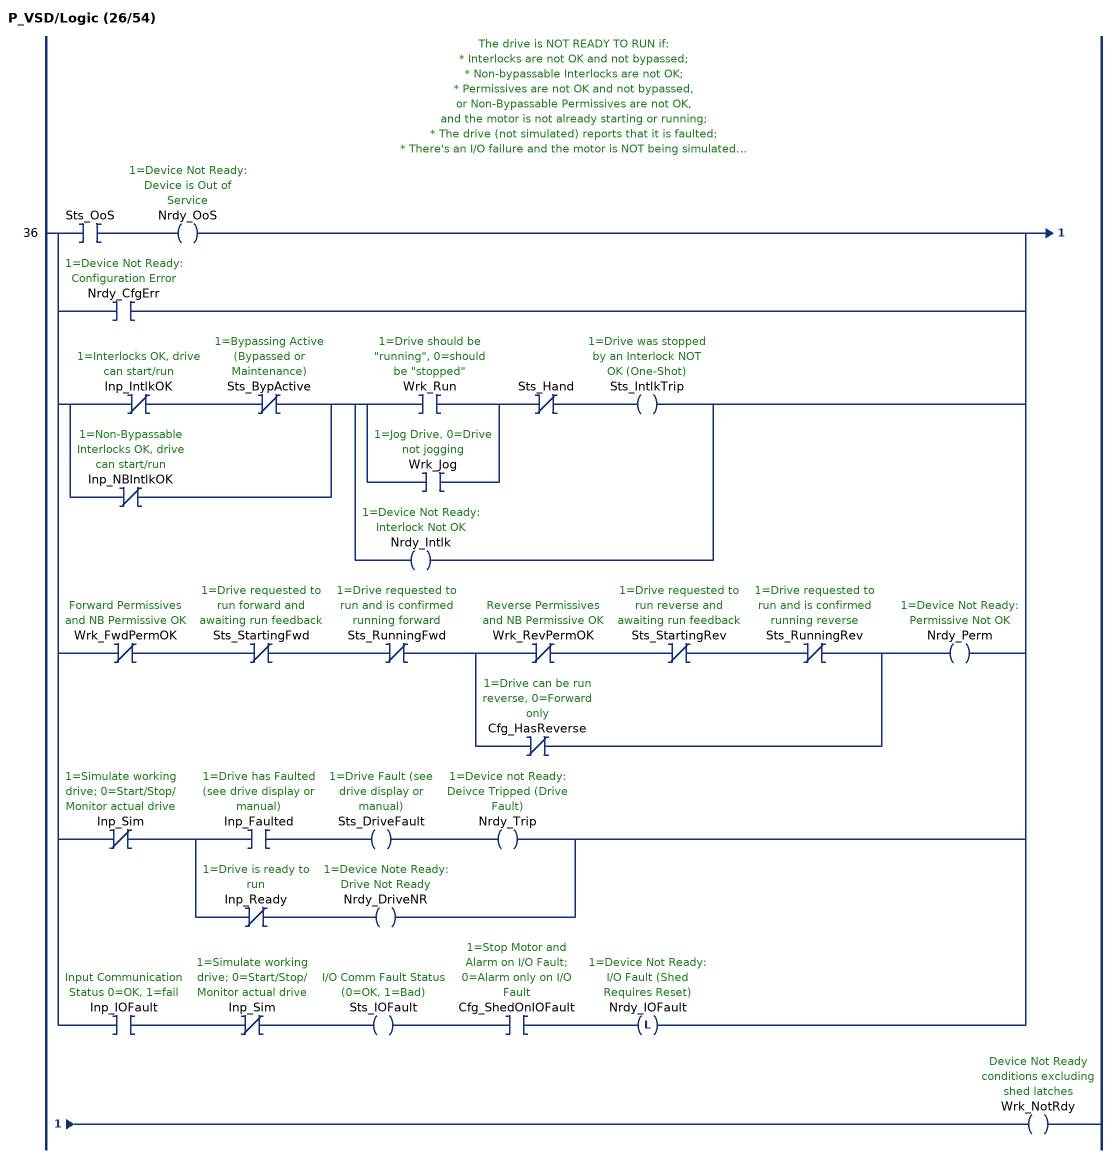
   // The drive is NOT READY TO RUN if:
   // * Interlocks are not OK and not bypassed;
   // * Non-bypassable Interlocks are not OK;
   // * Permissives are not OK and not bypassed,
   // or Non-Bypassable Permissives are not OK,
   // and the motor is not already starting or running;
   // * The drive (not simulated) reports that it is faulted;
   // * There's an I/O failure and the motor is NOT being simulated;
   // * The motor has a Fail to Start that has not been reset;
   // * The drive is disabled (by Maintenance);
   // * This instruction instance has a configuration error.
   // #####  V4.00.00  2018-07-13:  Disable/Enable replaced by P_CmdSrc Out of Service (OoS).  #####
   // #####  V4.00.00  2018-07-13:  Replaced start / stop / fwd / rev with start fwd / start rev / stop  #####
   36: [XIC(Sts_OoS) OTE(Nrdy_OoS) ,XIC(Nrdy_CfgErr) ,[XIO(Inp_IntlkOK) XIO(Sts_BypActive) ,XIO(Inp_NBIntlkOK) ] [[XIC(Wrk_Run) ,XIC(Wrk_Jog) ] XIO(Sts_Hand) OTE(Sts_IntlkTrip) ,OTE(Nrdy_Intlk) ] ,XIO(Wrk_FwdPermOK) XIO(Sts_StartingFwd) XIO(Sts_RunningFwd) [XIO(Wrk_RevPermOK) XIO(Sts_StartingRev) XIO(Sts_RunningRev) ,XIO(Cfg_HasReverse) ] OTE(Nrdy_Perm) ,XIO(Inp_Sim) [XIC(Inp_Faulted) OTE(Sts_DriveFault) OTE(Nrdy_Trip) ,XIO(Inp_Ready) OTE(Nrdy_DriveNR) ] ,XIC(Inp_IOFault) XIO(Inp_Sim) OTE(Sts_IOFault) XIC(Cfg_ShedOnIOFault) OTL(Nrdy_IOFault) ]OTE(Wrk_NotRdy);
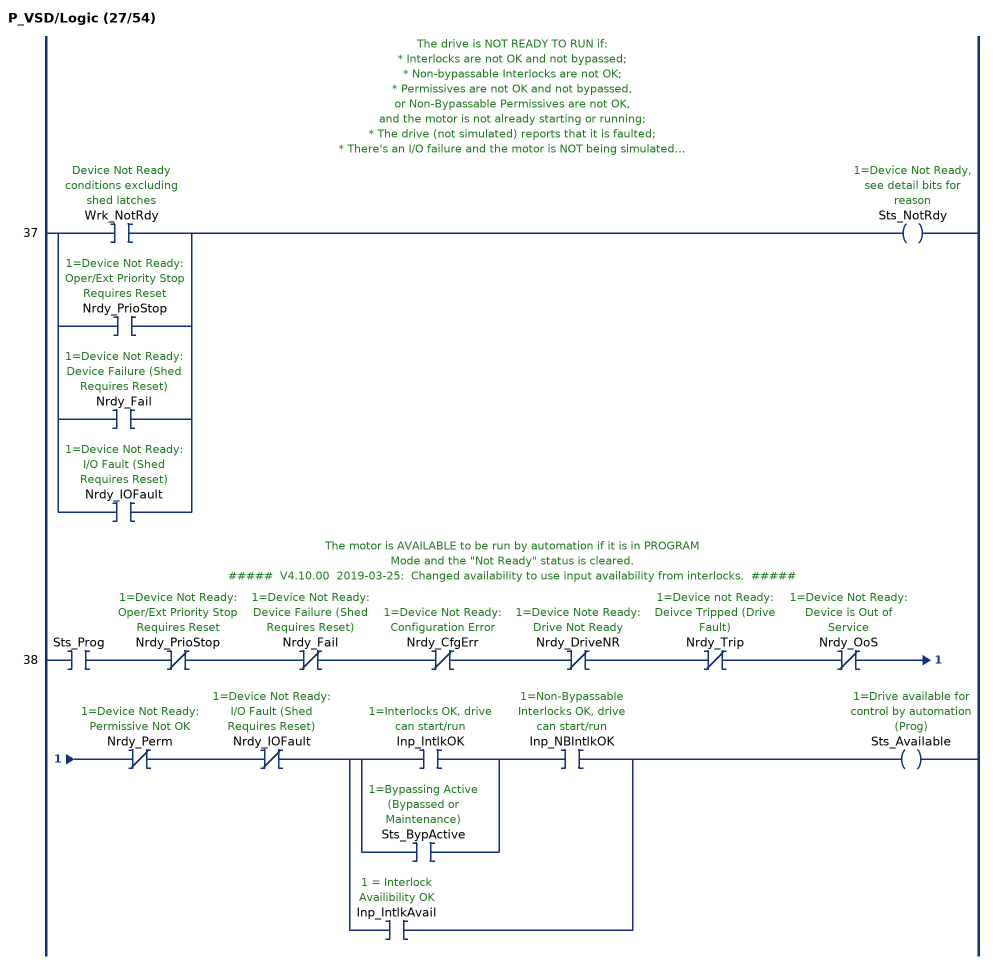
   // The drive is NOT READY TO RUN if:
   // * Interlocks are not OK and not bypassed;
   // * Non-bypassable Interlocks are not OK;
   // * Permissives are not OK and not bypassed,
   // or Non-Bypassable Permissives are not OK,
   // and the motor is not already starting or running;
   // * The drive (not simulated) reports that it is faulted;
   // * There's an I/O failure and the motor is NOT being simulated;
   // * The motor has a Fail to Start that has not been reset;
   // * The drive is disabled (by Maintenance);
   // * This instruction instance has a configuration error.
   37: [XIC(Wrk_NotRdy) ,XIC(Nrdy_PrioStop) ,XIC(Nrdy_Fail) ,XIC(Nrdy_IOFault) ]OTE(Sts_NotRdy);
   // The motor is AVAILABLE to be run by automation if it is in PROGRAM
   // Mode and the "Not Ready" status is cleared.
   // #####  V4.10.00  2019-03-25:  Changed availability to use input availability from interlocks.  #####
   38: XIC(Sts_Prog)XIO(Nrdy_PrioStop)XIO(Nrdy_Fail)XIO(Nrdy_CfgErr)XIO(Nrdy_DriveNR)XIO(Nrdy_Trip)XIO(Nrdy_OoS)XIO(Nrdy_Perm)XIO(Nrdy_IOFault)[[XIC(Inp_IntlkOK) ,XIC(Sts_BypActive) ] XIC(Inp_NBIntlkOK) ,XIC(Inp_IntlkAvail) ]OTE(Sts_Available);
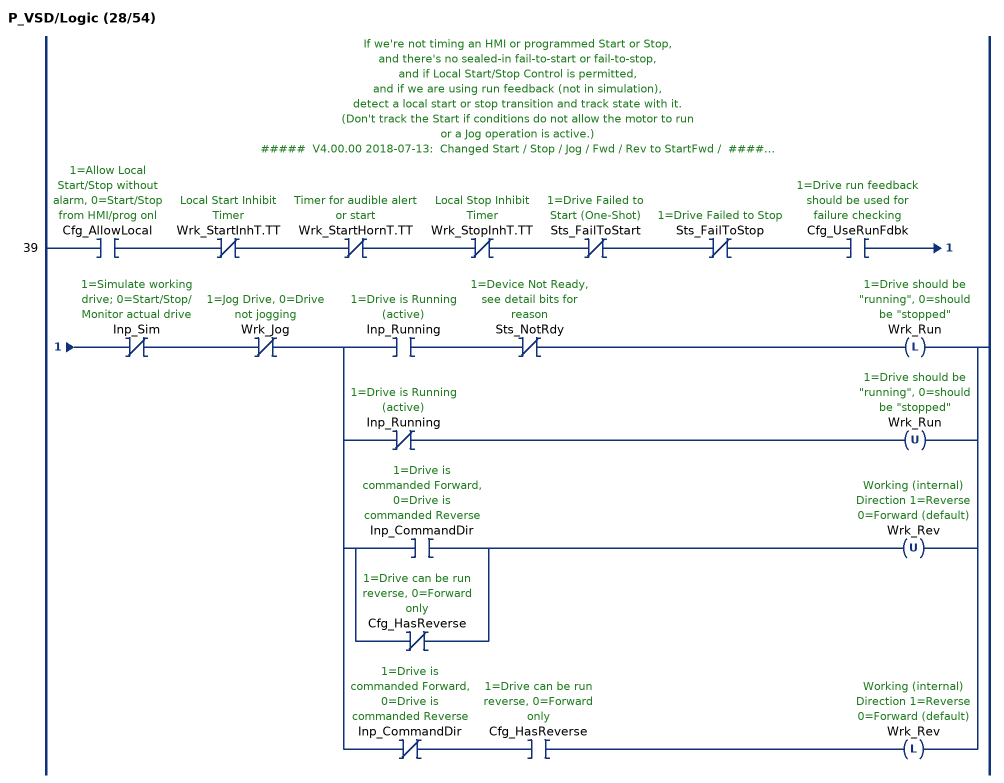
   // If we're not timing an HMI or programmed Start or Stop,
   // and there's no sealed-in fail-to-start or fail-to-stop,
   // and if Local Start/Stop Control is permitted,
   // and if we are using run feedback (not in simulation),
   // detect a local start or stop transition and track state with it.
   // (Don't track the Start if conditions do not allow the motor to run
   // or a Jog operation is active.)
   // #####  V4.00.00 2018-07-13:  Changed Start / Stop / Jog / Fwd / Rev to StartFwd /  #####
   // #####  StartRev / Stop / JogFwd / JogRev.  Deleted Cfg_PCmdClear.  #####
   // ##### V4.00.02  2018-10-30:  Corrected handling Allow Local when horn is enabled.  #####
   39: XIC(Cfg_AllowLocal)XIO(Wrk_StartInhT.TT)XIO(Wrk_StartHornT.TT)XIO(Wrk_StopInhT.TT)XIO(Sts_FailToStart)XIO(Sts_FailToStop)XIC(Cfg_UseRunFdbk)XIO(Inp_Sim)XIO(Wrk_Jog)[XIC(Inp_Running) XIO(Sts_NotRdy) OTL(Wrk_Run) ,XIO(Inp_Running) OTU(Wrk_Run) ,[XIC(Inp_CommandDir) ,XIO(Cfg_HasReverse) ] OTU(Wrk_Rev) ,XIO(Inp_CommandDir) XIC(Cfg_HasReverse) OTL(Wrk_Rev) ];
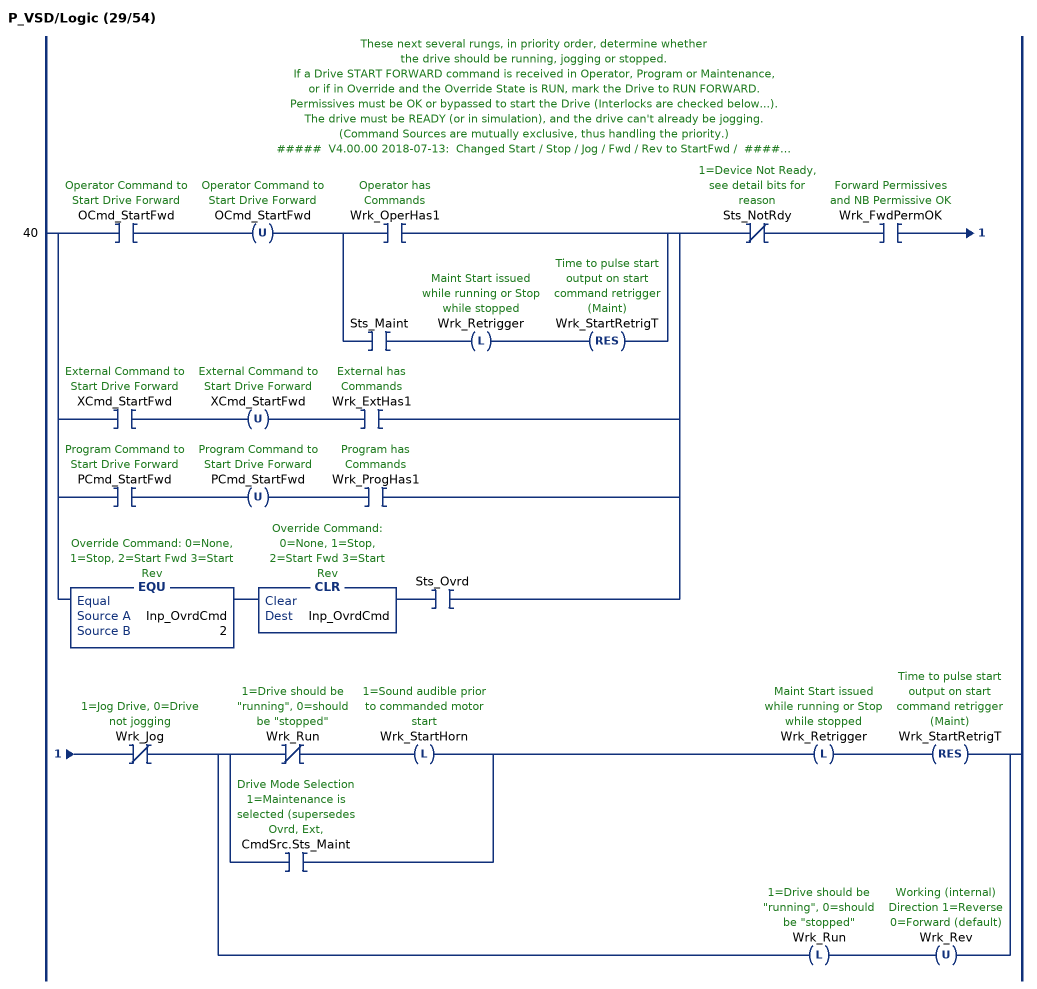
   // These next several rungs, in priority order, determine whether
   // the drive should be running, jogging or stopped.
   // If a Drive START FORWARD command is received in Operator, Program or Maintenance,
   // or if in Override and the Override State is RUN, mark the Drive to RUN FORWARD.
   // Permissives must be OK or bypassed to start the Drive (Interlocks are checked below...).
   // The drive must be READY (or in simulation), and the drive can't already be jogging.
   // (Command Sources are mutually exclusive, thus handling the priority.)
   // #####  V4.00.00 2018-07-13:  Changed Start / Stop / Jog / Fwd / Rev to StartFwd /  #####
   // #####  StartRev / Stop / JogFwd / JogRev.  Deleted Cfg_PCmdClear.  #####
   // #####  Added audible alert prior to commanded start.  #####
   // #####  Changed P_Mode to P_CmdSrc. Added External Command Source and Commands.  #####
   40: [XIC(OCmd_StartFwd) OTU(OCmd_StartFwd) [XIC(Wrk_OperHas1) ,XIC(Sts_Maint) OTL(Wrk_Retrigger) RES(Wrk_StartRetrigT) ] ,XIC(XCmd_StartFwd) OTU(XCmd_StartFwd) XIC(Wrk_ExtHas1) ,XIC(PCmd_StartFwd) OTU(PCmd_StartFwd) XIC(Wrk_ProgHas1) ,EQU(Inp_OvrdCmd,2) CLR(Inp_OvrdCmd) XIC(Sts_Ovrd) ]XIO(Sts_NotRdy)XIC(Wrk_FwdPermOK)XIO(Wrk_Jog)[[XIO(Wrk_Run) OTL(Wrk_StartHorn) ,XIC(CmdSrc.Sts_Maint) ] OTL(Wrk_Retrigger) RES(Wrk_StartRetrigT) ,OTL(Wrk_Run) OTU(Wrk_Rev) ];
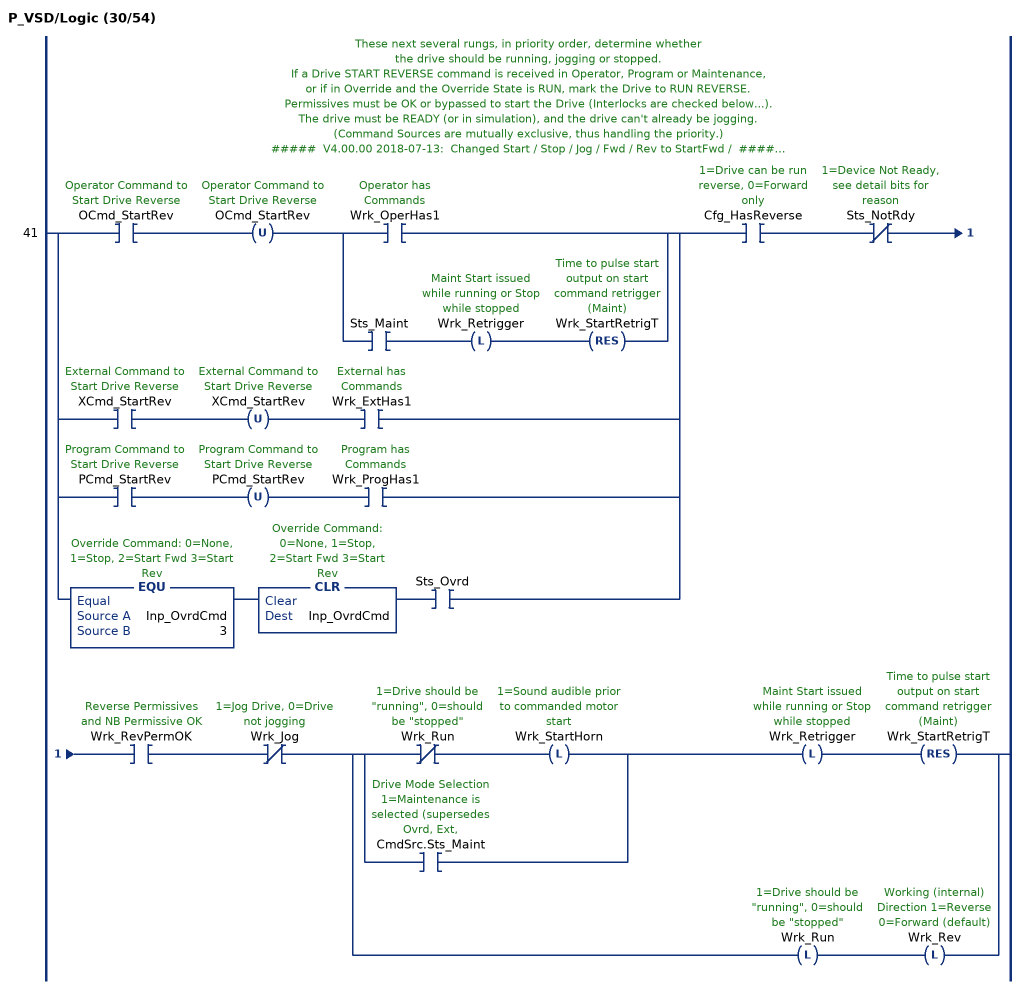
   // These next several rungs, in priority order, determine whether
   // the drive should be running, jogging or stopped.
   // If a Drive START REVERSE command is received in Operator, Program or Maintenance,
   // or if in Override and the Override State is RUN, mark the Drive to RUN REVERSE.
   // Permissives must be OK or bypassed to start the Drive (Interlocks are checked below...).
   // The drive must be READY (or in simulation), and the drive can't already be jogging.
   // (Command Sources are mutually exclusive, thus handling the priority.)
   // #####  V4.00.00 2018-07-13:  Changed Start / Stop / Jog / Fwd / Rev to StartFwd /  #####
   // #####  StartRev / Stop / JogFwd / JogRev.  Deleted Cfg_PCmdClear.  #####
   // #####  Added audible alert prior to commanded start.  #####
   // #####  Changed P_Mode to P_CmdSrc. Added External Command Source and Commands.  #####
   41: [XIC(OCmd_StartRev) OTU(OCmd_StartRev) [XIC(Wrk_OperHas1) ,XIC(Sts_Maint) OTL(Wrk_Retrigger) RES(Wrk_StartRetrigT) ] ,XIC(XCmd_StartRev) OTU(XCmd_StartRev) XIC(Wrk_ExtHas1) ,XIC(PCmd_StartRev) OTU(PCmd_StartRev) XIC(Wrk_ProgHas1) ,EQU(Inp_OvrdCmd,3) CLR(Inp_OvrdCmd) XIC(Sts_Ovrd) ]XIC(Cfg_HasReverse)XIO(Sts_NotRdy)XIC(Wrk_RevPermOK)XIO(Wrk_Jog)[[XIO(Wrk_Run) OTL(Wrk_StartHorn) ,XIC(CmdSrc.Sts_Maint) ] OTL(Wrk_Retrigger) RES(Wrk_StartRetrigT) ,OTL(Wrk_Run) OTL(Wrk_Rev) ];
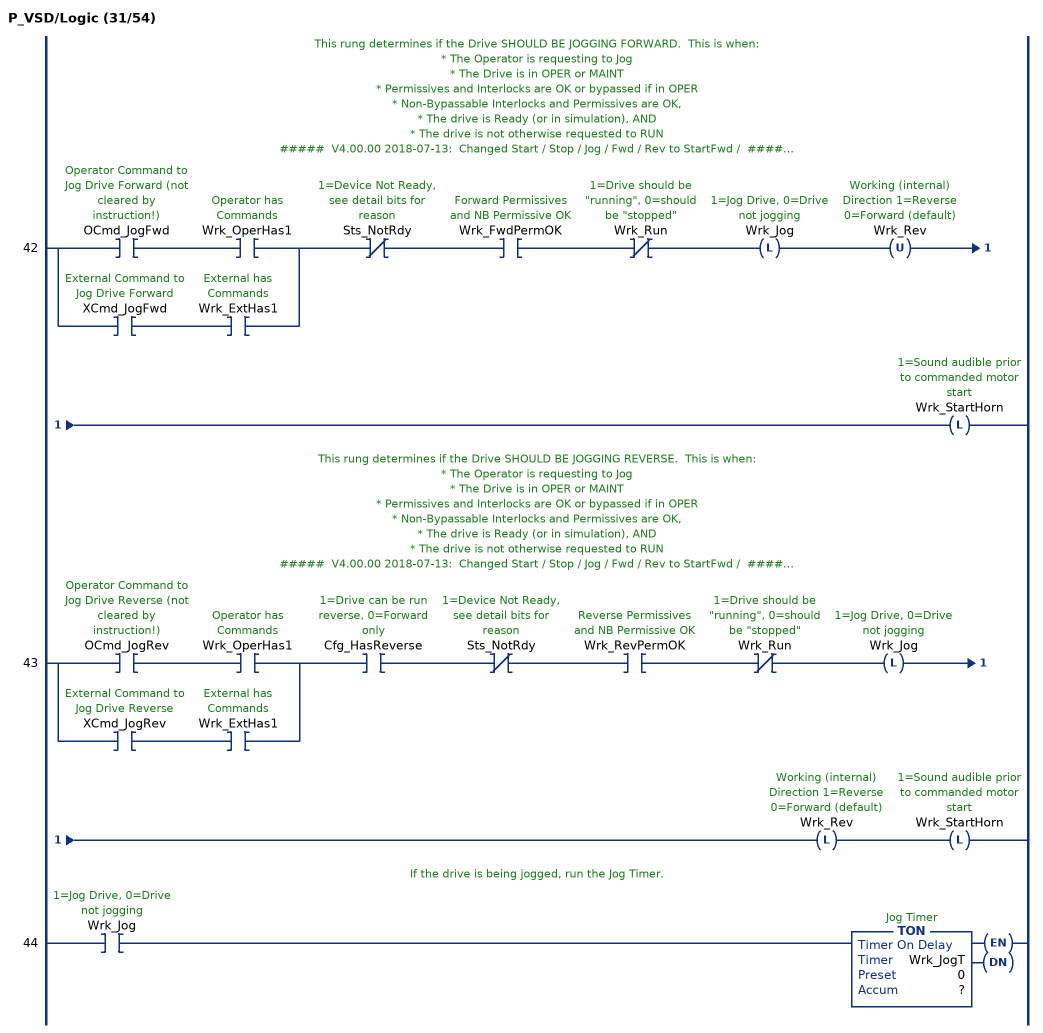
   // This rung determines if the Drive SHOULD BE JOGGING FORWARD.  This is when:
   // * The Operator is requesting to Jog
   // * The Drive is in OPER or MAINT
   // * Permissives and Interlocks are OK or bypassed if in OPER
   // * Non-Bypassable Interlocks and Permissives are OK,
   // * The drive is Ready (or in simulation), AND
   // * The drive is not otherwise requested to RUN
   // #####  V4.00.00 2018-07-13:  Changed Start / Stop / Jog / Fwd / Rev to StartFwd /  #####
   // #####  StartRev / Stop / JogFwd / JogRev.  Deleted Cfg_PCmdClear.  #####
   // #####  Changed P_Mode to P_CmdSrc. Added External Command Source and Commands.  #####
   42: [XIC(OCmd_JogFwd) XIC(Wrk_OperHas1) ,XIC(XCmd_JogFwd) XIC(Wrk_ExtHas1) ]XIO(Sts_NotRdy)XIC(Wrk_FwdPermOK)XIO(Wrk_Run)OTL(Wrk_Jog)OTU(Wrk_Rev)OTL(Wrk_StartHorn);
   // This rung determines if the Drive SHOULD BE JOGGING REVERSE.  This is when:
   // * The Operator is requesting to Jog
   // * The Drive is in OPER or MAINT
   // * Permissives and Interlocks are OK or bypassed if in OPER
   // * Non-Bypassable Interlocks and Permissives are OK,
   // * The drive is Ready (or in simulation), AND
   // * The drive is not otherwise requested to RUN
   // #####  V4.00.00 2018-07-13:  Changed Start / Stop / Jog / Fwd / Rev to StartFwd /  #####
   // #####  StartRev / Stop / JogFwd / JogRev.  Deleted Cfg_PCmdClear.  #####
   // #####  Changed P_Mode to P_CmdSrc. Added External Command Source and Commands.  #####
   43: [XIC(OCmd_JogRev) XIC(Wrk_OperHas1) ,XIC(XCmd_JogRev) XIC(Wrk_ExtHas1) ]XIC(Cfg_HasReverse)XIO(Sts_NotRdy)XIC(Wrk_RevPermOK)XIO(Wrk_Run)OTL(Wrk_Jog)OTL(Wrk_Rev)OTL(Wrk_StartHorn);
   // If the drive is being jogged, run the Jog Timer.
   44: XIC(Wrk_Jog)TON(Wrk_JogT,?,?);
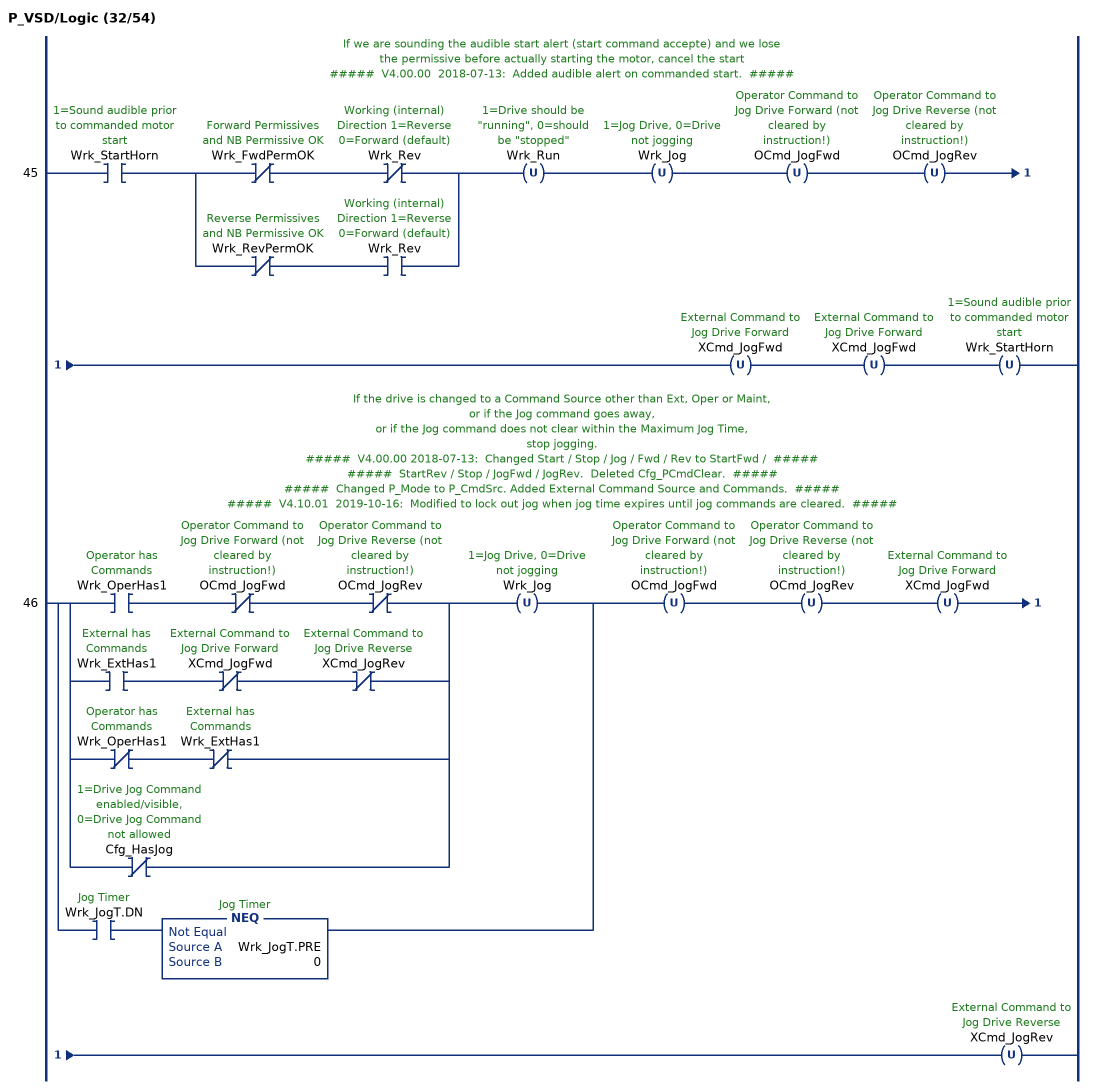
   // If we are sounding the audible start alert (start command accepte) and we lose
   // the permissive before actually starting the motor, cancel the start
   // #####  V4.00.00  2018-07-13:  Added audible alert on commanded start.  #####
   45: XIC(Wrk_StartHorn)[XIO(Wrk_FwdPermOK) XIO(Wrk_Rev) ,XIO(Wrk_RevPermOK) XIC(Wrk_Rev) ]OTU(Wrk_Run)OTU(Wrk_Jog)OTU(OCmd_JogFwd)OTU(OCmd_JogRev)OTU(XCmd_JogFwd)OTU(XCmd_JogFwd)OTU(Wrk_StartHorn);
   // If the drive is changed to a Command Source other than Ext, Oper or Maint,
   // or if the Jog command goes away,
   // or if the Jog command does not clear within the Maximum Jog Time,
   // stop jogging.
   // #####  V4.00.00 2018-07-13:  Changed Start / Stop / Jog / Fwd / Rev to StartFwd /  #####
   // #####  StartRev / Stop / JogFwd / JogRev.  Deleted Cfg_PCmdClear.  #####
   // #####  Changed P_Mode to P_CmdSrc. Added External Command Source and Commands.  #####
   // #####  V4.10.01  2019-10-16:  Modified to lock out jog when jog time expires until jog commands are cleared.  #####
   46: [[XIC(Wrk_OperHas1) XIO(OCmd_JogFwd) XIO(OCmd_JogRev) ,XIC(Wrk_ExtHas1) XIO(XCmd_JogFwd) XIO(XCmd_JogRev) ,XIO(Wrk_OperHas1) XIO(Wrk_ExtHas1) ,XIO(Cfg_HasJog) ] OTU(Wrk_Jog) ,XIC(Wrk_JogT.DN) NEQ(Wrk_JogT.PRE,0) ]OTU(OCmd_JogFwd)OTU(OCmd_JogRev)OTU(XCmd_JogFwd)OTU(XCmd_JogRev);
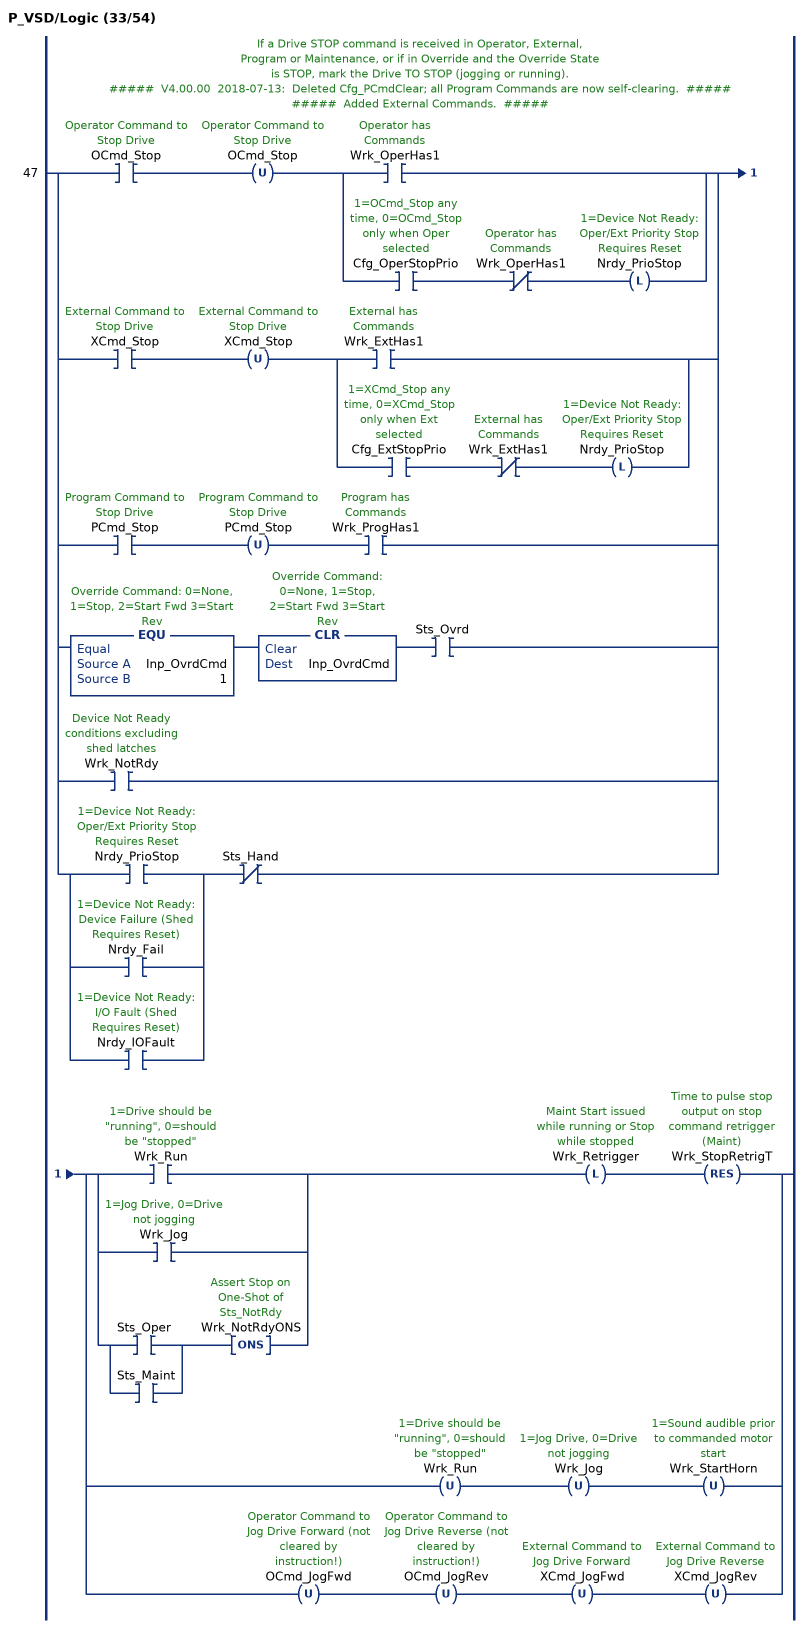
   // If a Drive STOP command is received in Operator, External,
   // Program or Maintenance, or if in Override and the Override State
   // is STOP, mark the Drive TO STOP (jogging or running).
   // #####  V4.00.00  2018-07-13:  Deleted Cfg_PCmdClear; all Program Commands are now self-clearing.  #####
   // #####  Added External Commands.  #####
   47: [XIC(OCmd_Stop) OTU(OCmd_Stop) [XIC(Wrk_OperHas1) ,XIC(Cfg_OperStopPrio) XIO(Wrk_OperHas1) OTL(Nrdy_PrioStop) ] ,XIC(XCmd_Stop) OTU(XCmd_Stop) [XIC(Wrk_ExtHas1) ,XIC(Cfg_ExtStopPrio) XIO(Wrk_ExtHas1) OTL(Nrdy_PrioStop) ] ,XIC(PCmd_Stop) OTU(PCmd_Stop) XIC(Wrk_ProgHas1) ,EQU(Inp_OvrdCmd,1) CLR(Inp_OvrdCmd) XIC(Sts_Ovrd) ,XIC(Wrk_NotRdy) ,[XIC(Nrdy_PrioStop) ,XIC(Nrdy_Fail) ,XIC(Nrdy_IOFault) ] XIO(Sts_Hand) ][[XIC(Wrk_Run) ,XIC(Wrk_Jog) ,[XIC(Sts_Oper) ,XIC(Sts_Maint) ] ONS(Wrk_NotRdyONS) ] OTL(Wrk_Retrigger) RES(Wrk_StopRetrigT) ,OTU(Wrk_Run) OTU(Wrk_Jog) OTU(Wrk_StartHorn) ,OTU(OCmd_JogFwd) OTU(OCmd_JogRev) OTU(XCmd_JogFwd) OTU(XCmd_JogRev) ];
